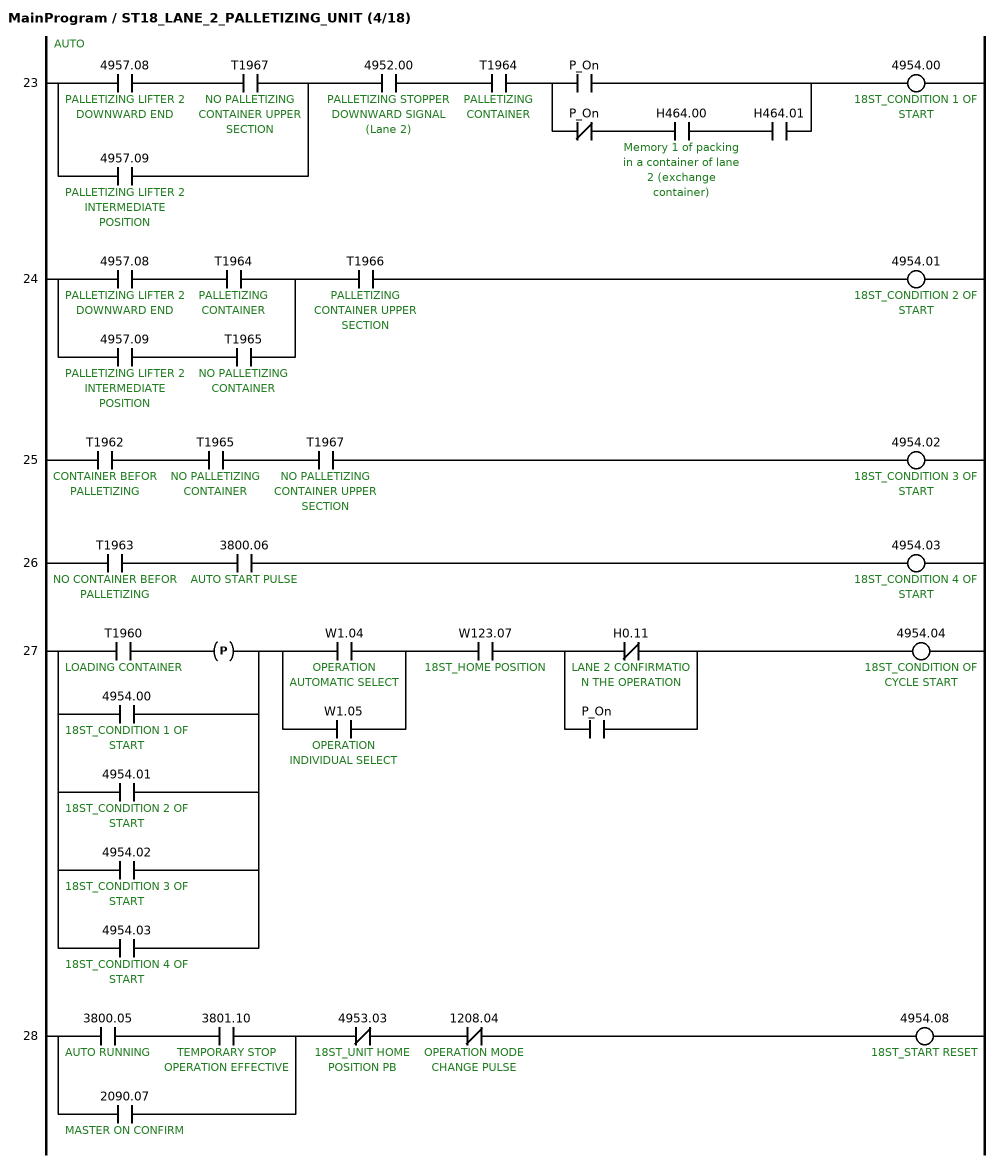
; [picture p672: MainProgram / ST18_LANE_2_PALLETIZING_UNIT, rungs 23-28]
; rung 23: AUTO
LD 4957.08  ; PALLETIZING LIFTER 2 DOWNWARD END
AND T1967  ; NO PALLETIZING CONTAINER UPPER SECTION
OR 4957.09  ; PALLETIZING LIFTER 2 INTERMEDIATE POSITION
AND 4952.00  ; PALLETIZING STOPPER DOWNWARD SIGNAL (Lane 2)
AND T1964  ; PALLETIZING CONTAINER
LD P_On
LDNOT P_On
AND H464.00  ; Memory 1 of packing in a container of lane 2 (exchange container)
AND H464.01
ORLD
ANDLD
OUT 4954.00  ; 18ST_CONDITION 1 OF START
; rung 24
LD 4957.08  ; PALLETIZING LIFTER 2 DOWNWARD END
AND T1964  ; PALLETIZING CONTAINER
LD 4957.09  ; PALLETIZING LIFTER 2 INTERMEDIATE POSITION
AND T1965  ; NO PALLETIZING CONTAINER
ORLD
AND T1966  ; PALLETIZING CONTAINER UPPER SECTION
OUT 4954.01  ; 18ST_CONDITION 2 OF START
; rung 25
LD T1962  ; CONTAINER BEFOR PALLETIZING
AND T1965  ; NO PALLETIZING CONTAINER
AND T1967  ; NO PALLETIZING CONTAINER UPPER SECTION
OUT 4954.02  ; 18ST_CONDITION 3 OF START
; rung 26
LD T1963  ; NO CONTAINER BEFOR PALLETIZING
AND 3800.06  ; AUTO START PULSE
OUT 4954.03  ; 18ST_CONDITION 4 OF START
; rung 27
LD T1960  ; LOADING CONTAINER
UP(521)
OR 4954.00  ; 18ST_CONDITION 1 OF START
OR 4954.01  ; 18ST_CONDITION 2 OF START
OR 4954.02  ; 18ST_CONDITION 3 OF START
OR 4954.03  ; 18ST_CONDITION 4 OF START
LD W1.04  ; OPERATION AUTOMATIC SELECT
OR W1.05  ; OPERATION INDIVIDUAL SELECT
ANDLD
AND W123.07  ; 18ST_HOME POSITION
LDNOT H0.11  ; LANE 2 CONFIRMATION THE OPERATION
OR P_On
ANDLD
OUT 4954.04  ; 18ST_CONDITION OF CYCLE START
; rung 28
LD 3800.05  ; AUTO RUNNING
AND 3801.10  ; TEMPORARY STOP OPERATION EFFECTIVE
OR 2090.07  ; MASTER ON CONFIRM
ANDNOT 4953.03  ; 18ST_UNIT HOME POSITION PB
ANDNOT 1208.04  ; OPERATION MODE CHANGE PULSE
OUT 4954.08  ; 18ST_START RESET

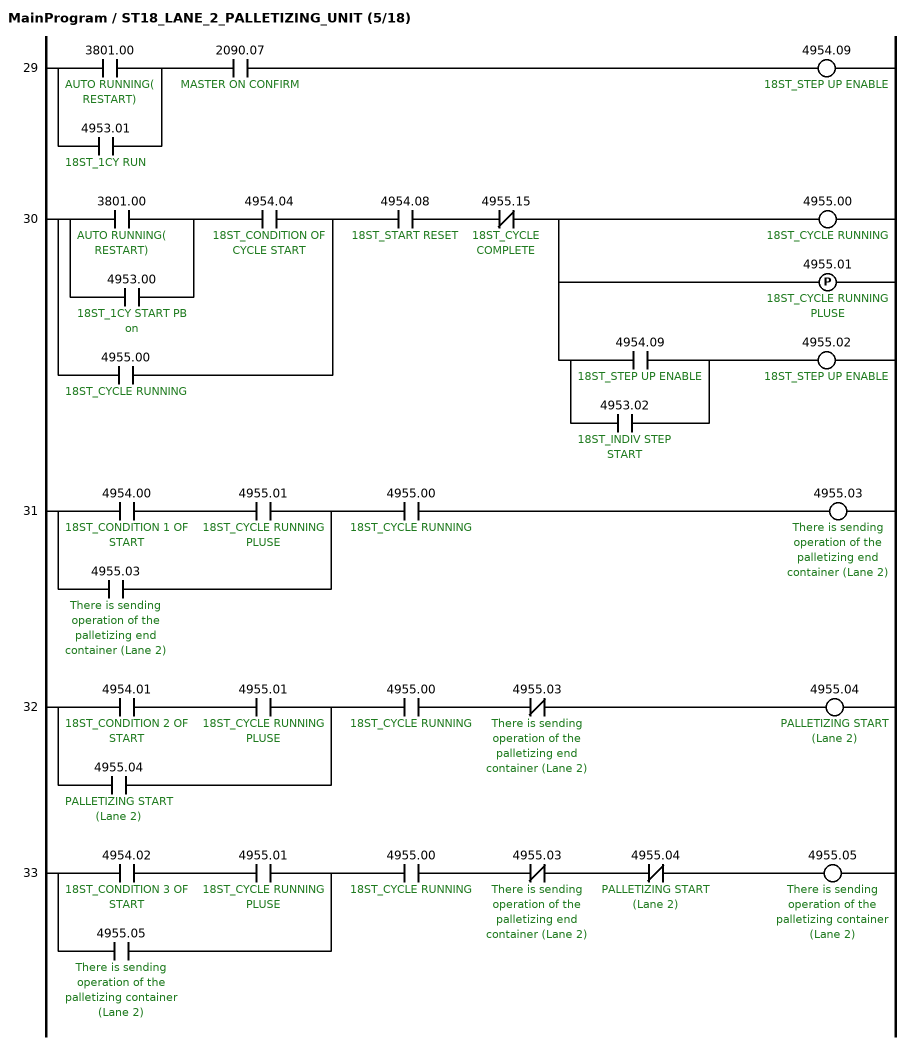
; rung 29
LD 3801.00  ; AUTO RUNNING(RESTART)
OR 4953.01  ; 18ST_1CY RUN
AND 2090.07  ; MASTER ON CONFIRM
OUT 4954.09  ; 18ST_STEP UP ENABLE
; rung 30
LD 3801.00  ; AUTO RUNNING(RESTART)
OR 4953.00  ; 18ST_1CY START PB on
AND 4954.04  ; 18ST_CONDITION OF CYCLE START
OR 4955.00  ; 18ST_CYCLE RUNNING
AND 4954.08  ; 18ST_START RESET
ANDNOT 4955.15  ; 18ST_CYCLE COMPLETE
OUT 4955.00  ; 18ST_CYCLE RUNNING
DIFU(013) 4955.01  ; 18ST_CYCLE RUNNING PLUSE
LD 4954.09  ; 18ST_STEP UP ENABLE
OR 4953.02  ; 18ST_INDIV STEP START
ANDLD
OUT 4955.02  ; 18ST_STEP UP ENABLE
; rung 31
LD 4954.00  ; 18ST_CONDITION 1 OF START
AND 4955.01  ; 18ST_CYCLE RUNNING PLUSE
OR 4955.03  ; There is sending operation of the palletizing end container (Lane 2)
AND 4955.00  ; 18ST_CYCLE RUNNING
OUT 4955.03  ; There is sending operation of the palletizing end container (Lane 2)
; rung 32
LD 4954.01  ; 18ST_CONDITION 2 OF START
AND 4955.01  ; 18ST_CYCLE RUNNING PLUSE
OR 4955.04  ; PALLETIZING START (Lane 2)
AND 4955.00  ; 18ST_CYCLE RUNNING
ANDNOT 4955.03  ; There is sending operation of the palletizing end container (Lane 2)
OUT 4955.04  ; PALLETIZING START (Lane 2)
; rung 33
LD 4954.02  ; 18ST_CONDITION 3 OF START
AND 4955.01  ; 18ST_CYCLE RUNNING PLUSE
OR 4955.05  ; There is sending operation of the palletizing container (Lane 2)
AND 4955.00  ; 18ST_CYCLE RUNNING
ANDNOT 4955.03  ; There is sending operation of the palletizing end container (Lane 2)
ANDNOT 4955.04  ; PALLETIZING START (Lane 2)
OUT 4955.05  ; There is sending operation of the palletizing container (Lane 2)

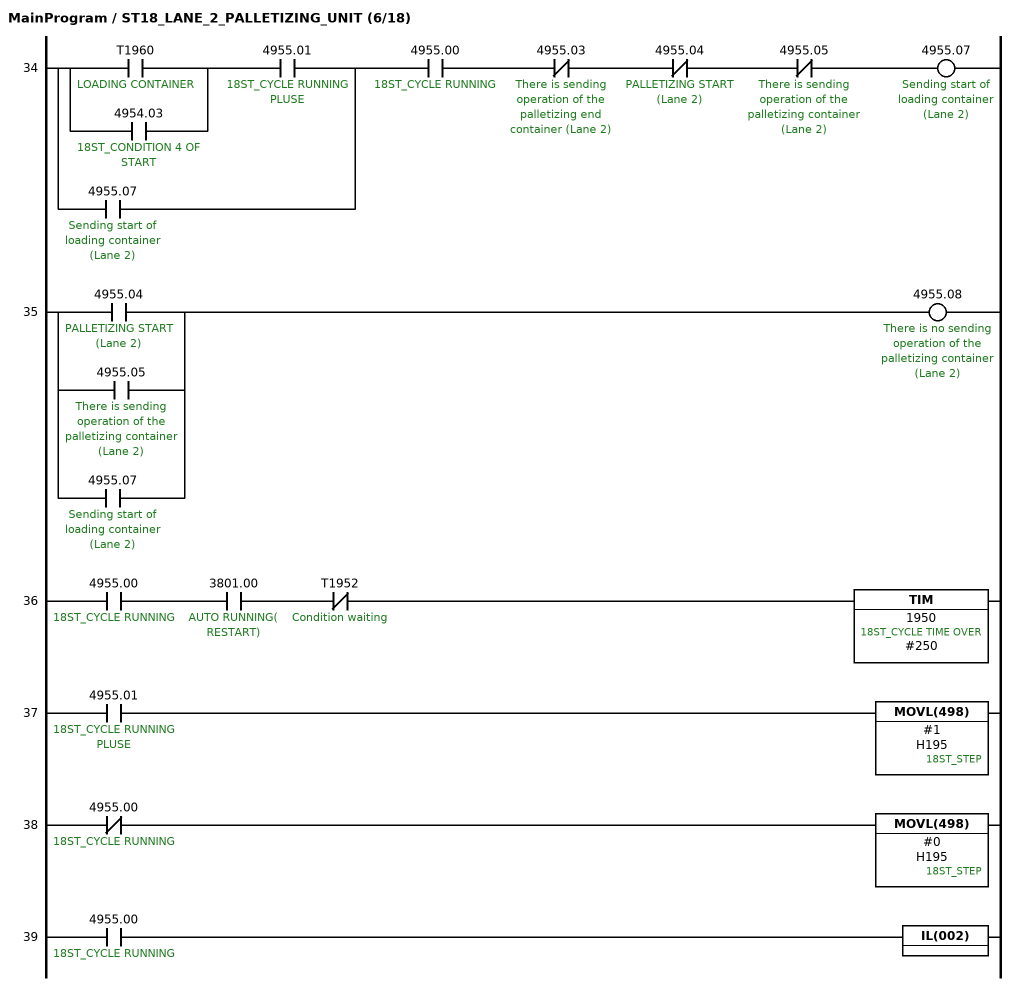
; rung 34
LD T1960  ; LOADING CONTAINER
OR 4954.03  ; 18ST_CONDITION 4 OF START
AND 4955.01  ; 18ST_CYCLE RUNNING PLUSE
OR 4955.07  ; Sending start of loading container (Lane 2)
AND 4955.00  ; 18ST_CYCLE RUNNING
ANDNOT 4955.03  ; There is sending operation of the palletizing end container (Lane 2)
ANDNOT 4955.04  ; PALLETIZING START (Lane 2)
ANDNOT 4955.05  ; There is sending operation of the palletizing container (Lane 2)
OUT 4955.07  ; Sending start of loading container (Lane 2)
; rung 35
LD 4955.04  ; PALLETIZING START (Lane 2)
OR 4955.05  ; There is sending operation of the palletizing container (Lane 2)
OR 4955.07  ; Sending start of loading container (Lane 2)
OUT 4955.08  ; There is no sending operation of the palletizing container (Lane 2)
; rung 36
LD 4955.00  ; 18ST_CYCLE RUNNING
AND 3801.00  ; AUTO RUNNING(RESTART)
ANDNOT T1952  ; Condition waiting
TIM 1950 #250  ; 18ST_CYCLE TIME OVER
; rung 37
LD 4955.01  ; 18ST_CYCLE RUNNING PLUSE
MOVL(498) #1 H195  ; 18ST_STEP
; rung 38
LDNOT 4955.00  ; 18ST_CYCLE RUNNING
MOVL(498) #0 H195  ; 18ST_STEP
; rung 39
LD 4955.00  ; 18ST_CYCLE RUNNING
IL(002)

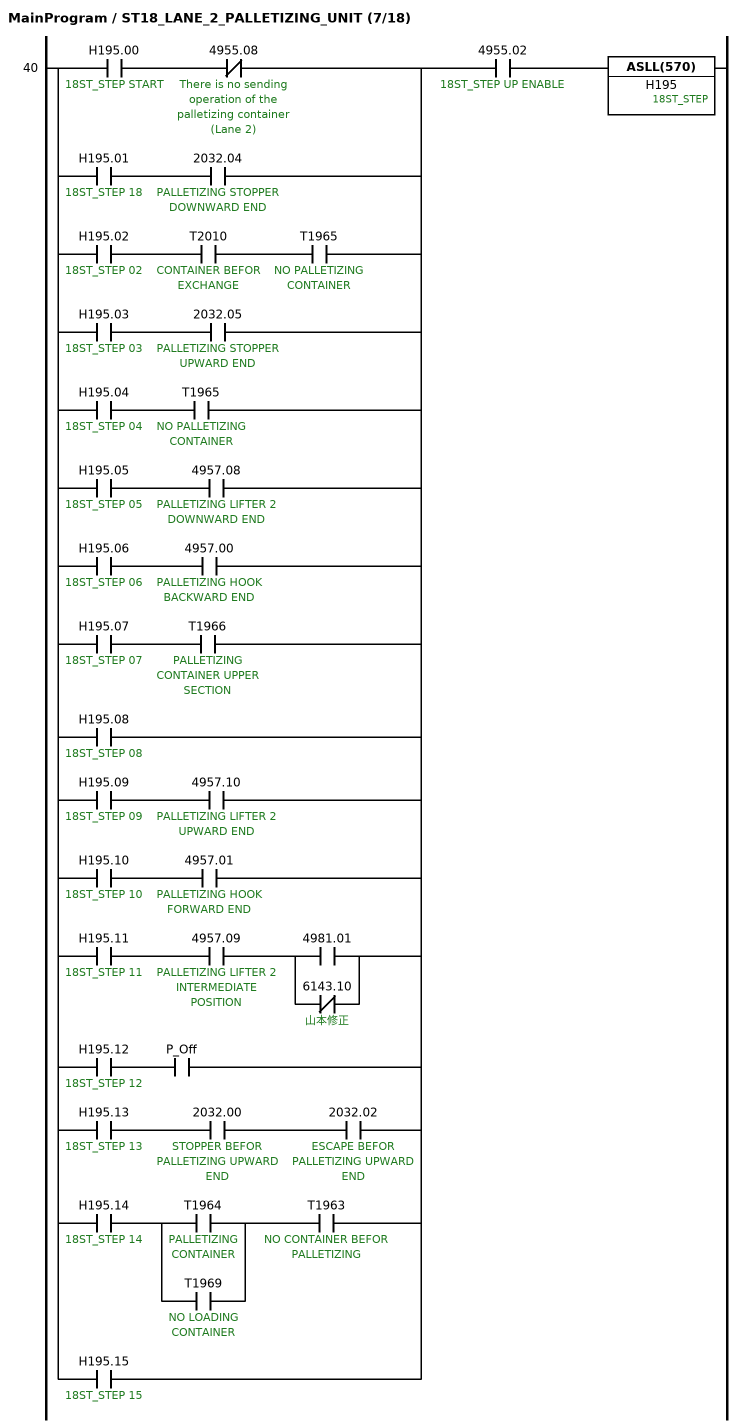
; rung 40
LD H195.00  ; 18ST_STEP START
ANDNOT 4955.08  ; There is no sending operation of the palletizing container (Lane 2)
LD H195.01  ; 18ST_STEP 18
AND 2032.04  ; PALLETIZING STOPPER DOWNWARD END
ORLD
LD H195.02  ; 18ST_STEP 02
AND T2010  ; CONTAINER BEFOR EXCHANGE
AND T1965  ; NO PALLETIZING CONTAINER
ORLD
LD H195.03  ; 18ST_STEP 03
AND 2032.05  ; PALLETIZING STOPPER UPWARD END
ORLD
LD H195.04  ; 18ST_STEP 04
AND T1965  ; NO PALLETIZING CONTAINER
ORLD
LD H195.05  ; 18ST_STEP 05
AND 4957.08  ; PALLETIZING LIFTER 2 DOWNWARD END
ORLD
LD H195.06  ; 18ST_STEP 06
AND 4957.00  ; PALLETIZING HOOK BACKWARD END
ORLD
LD H195.07  ; 18ST_STEP 07
AND T1966  ; PALLETIZING CONTAINER UPPER SECTION
ORLD
OR H195.08  ; 18ST_STEP 08
LD H195.09  ; 18ST_STEP 09
AND 4957.10  ; PALLETIZING LIFTER 2 UPWARD END
ORLD
LD H195.10  ; 18ST_STEP 10
AND 4957.01  ; PALLETIZING HOOK FORWARD END
ORLD
LD H195.11  ; 18ST_STEP 11
AND 4957.09  ; PALLETIZING LIFTER 2 INTERMEDIATE POSITION
LD 4981.01
ORNOT 6143.10  ; 山本修正
ANDLD
ORLD
LD H195.12  ; 18ST_STEP 12
AND P_Off
ORLD
LD H195.13  ; 18ST_STEP 13
AND 2032.00  ; STOPPER BEFOR PALLETIZING UPWARD END
AND 2032.02  ; ESCAPE BEFOR PALLETIZING UPWARD END
ORLD
LD H195.14  ; 18ST_STEP 14
LD T1964  ; PALLETIZING CONTAINER
OR T1969  ; NO LOADING CONTAINER
ANDLD
AND T1963  ; NO CONTAINER BEFOR PALLETIZING
ORLD
OR H195.15  ; 18ST_STEP 15
AND 4955.02  ; 18ST_STEP UP ENABLE
ASLL(570) H195  ; 18ST_STEP

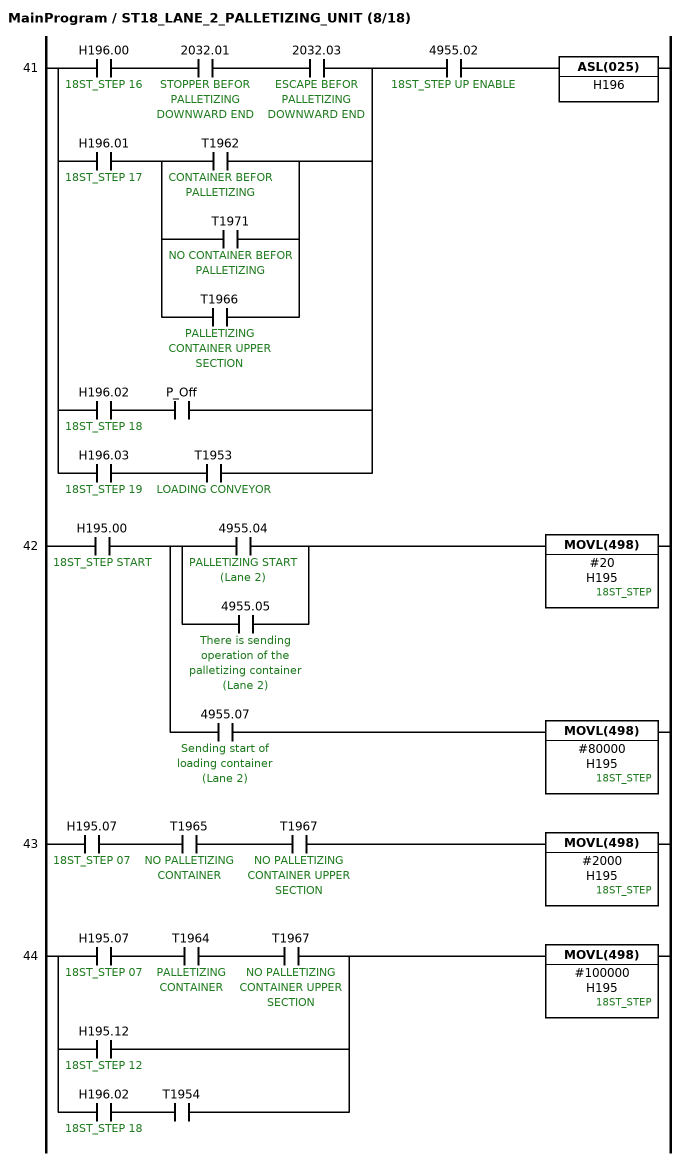
; rung 41
LD H196.00  ; 18ST_STEP 16
AND 2032.01  ; STOPPER BEFOR PALLETIZING DOWNWARD END
AND 2032.03  ; ESCAPE BEFOR PALLETIZING DOWNWARD END
LD H196.01  ; 18ST_STEP 17
LD T1962  ; CONTAINER BEFOR PALLETIZING
OR T1971  ; NO CONTAINER BEFOR PALLETIZING
OR T1966  ; PALLETIZING CONTAINER UPPER SECTION
ANDLD
ORLD
LD H196.02  ; 18ST_STEP 18
AND P_Off
ORLD
LD H196.03  ; 18ST_STEP 19
AND T1953  ; LOADING CONVEYOR
ORLD
AND 4955.02  ; 18ST_STEP UP ENABLE
ASL(025) H196
; rung 42
LD H195.00  ; 18ST_STEP START
OUT TR0
LD 4955.04  ; PALLETIZING START (Lane 2)
OR 4955.05  ; There is sending operation of the palletizing container (Lane 2)
ANDLD
MOVL(498) #20 H195  ; 18ST_STEP
LD TR0
AND 4955.07  ; Sending start of loading container (Lane 2)
MOVL(498) #80000 H195  ; 18ST_STEP
; rung 43
LD H195.07  ; 18ST_STEP 07
AND T1965  ; NO PALLETIZING CONTAINER
AND T1967  ; NO PALLETIZING CONTAINER UPPER SECTION
MOVL(498) #2000 H195  ; 18ST_STEP
; rung 44
LD H195.07  ; 18ST_STEP 07
AND T1964  ; PALLETIZING CONTAINER
AND T1967  ; NO PALLETIZING CONTAINER UPPER SECTION
OR H195.12  ; 18ST_STEP 12
LD H196.02  ; 18ST_STEP 18
AND T1954
ORLD
MOVL(498) #100000 H195  ; 18ST_STEP

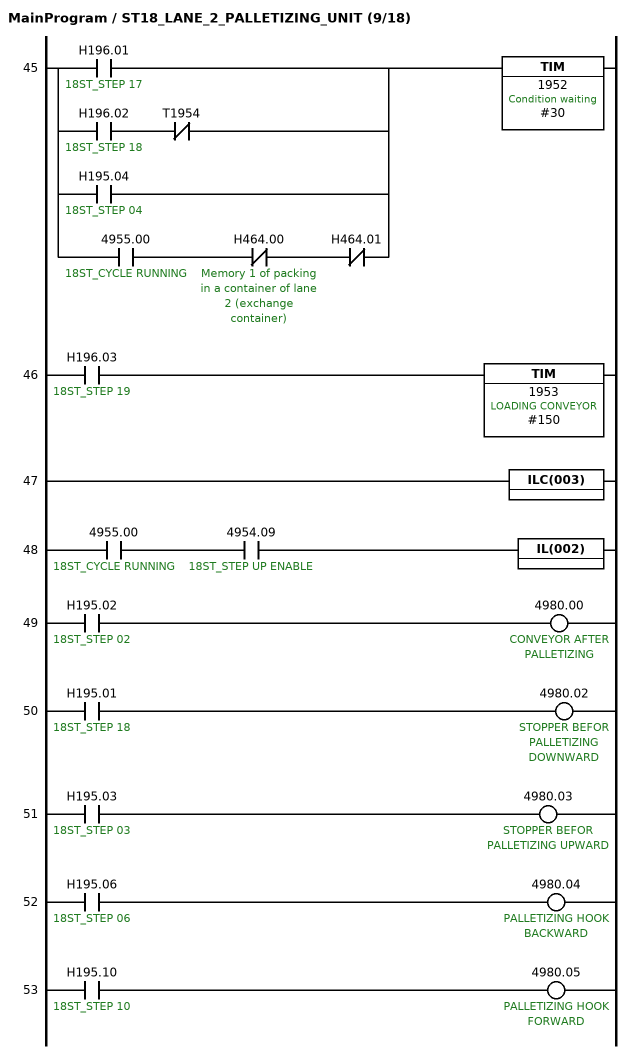
; rung 45
LD H196.01  ; 18ST_STEP 17
LD H196.02  ; 18ST_STEP 18
ANDNOT T1954
ORLD
OR H195.04  ; 18ST_STEP 04
LD 4955.00  ; 18ST_CYCLE RUNNING
ANDNOT H464.00  ; Memory 1 of packing in a container of lane 2 (exchange container)
ANDNOT H464.01
ORLD
TIM 1952 #30  ; Condition waiting
; rung 46
LD H196.03  ; 18ST_STEP 19
TIM 1953 #150  ; LOADING CONVEYOR
; rung 47
ILC(003)
; rung 48
LD 4955.00  ; 18ST_CYCLE RUNNING
AND 4954.09  ; 18ST_STEP UP ENABLE
IL(002)
; rung 49
LD H195.02  ; 18ST_STEP 02
OUT 4980.00  ; CONVEYOR AFTER PALLETIZING
; rung 50
LD H195.01  ; 18ST_STEP 18
OUT 4980.02  ; STOPPER BEFOR PALLETIZING DOWNWARD
; rung 51
LD H195.03  ; 18ST_STEP 03
OUT 4980.03  ; STOPPER BEFOR PALLETIZING UPWARD
; rung 52
LD H195.06  ; 18ST_STEP 06
OUT 4980.04  ; PALLETIZING HOOK BACKWARD
; rung 53
LD H195.10  ; 18ST_STEP 10
OUT 4980.05  ; PALLETIZING HOOK FORWARD

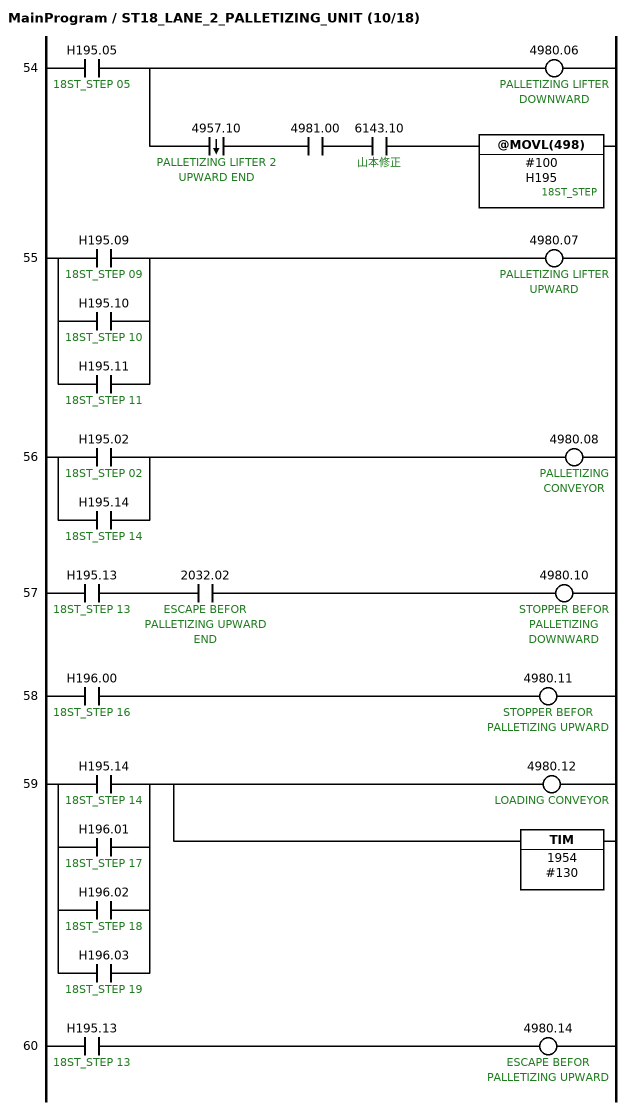
; rung 54
LD H195.05  ; 18ST_STEP 05
OUT 4980.06  ; PALLETIZING LIFTER DOWNWARD
%AND 4957.10  ; PALLETIZING LIFTER 2 UPWARD END
AND 4981.00
AND 6143.10  ; 山本修正
@MOVL(498) #100 H195  ; 18ST_STEP
; rung 55
LD H195.09  ; 18ST_STEP 09
OR H195.10  ; 18ST_STEP 10
OR H195.11  ; 18ST_STEP 11
OUT 4980.07  ; PALLETIZING LIFTER UPWARD
; rung 56
LD H195.02  ; 18ST_STEP 02
OR H195.14  ; 18ST_STEP 14
OUT 4980.08  ; PALLETIZING CONVEYOR
; rung 57
LD H195.13  ; 18ST_STEP 13
AND 2032.02  ; ESCAPE BEFOR PALLETIZING UPWARD END
OUT 4980.10  ; STOPPER BEFOR PALLETIZING DOWNWARD
; rung 58
LD H196.00  ; 18ST_STEP 16
OUT 4980.11  ; STOPPER BEFOR PALLETIZING UPWARD
; rung 59
LD H195.14  ; 18ST_STEP 14
OR H196.01  ; 18ST_STEP 17
OR H196.02  ; 18ST_STEP 18
OR H196.03  ; 18ST_STEP 19
OUT 4980.12  ; LOADING CONVEYOR
TIM 1954 #130
; rung 60
LD H195.13  ; 18ST_STEP 13
OUT 4980.14  ; ESCAPE BEFOR PALLETIZING UPWARD

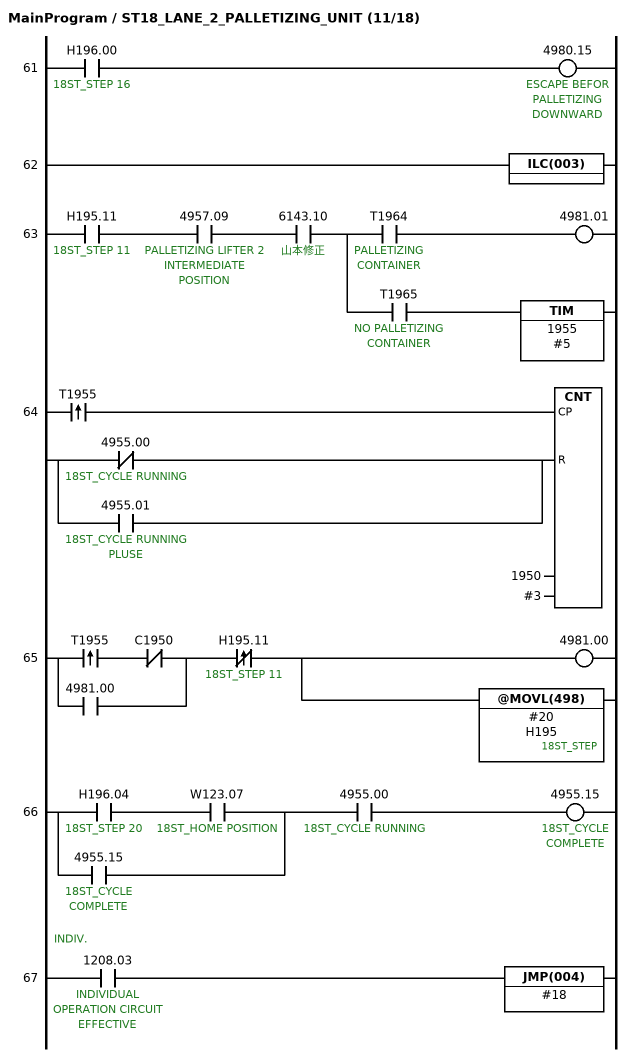
; rung 61
LD H196.00  ; 18ST_STEP 16
OUT 4980.15  ; ESCAPE BEFOR PALLETIZING DOWNWARD
; rung 62
ILC(003)
; rung 63
LD H195.11  ; 18ST_STEP 11
AND 4957.09  ; PALLETIZING LIFTER 2 INTERMEDIATE POSITION
AND 6143.10  ; 山本修正
OUT TR0
AND T1964  ; PALLETIZING CONTAINER
OUT 4981.01
LD TR0
AND T1965  ; NO PALLETIZING CONTAINER
TIM 1955 #5
; rung 64
@LD T1955
LDNOT 4955.00  ; 18ST_CYCLE RUNNING
OR 4955.01  ; 18ST_CYCLE RUNNING PLUSE
CNT 1950 #3
; rung 65
@LD T1955
ANDNOT C1950
OR 4981.00
@ANDNOT H195.11  ; 18ST_STEP 11
OUT 4981.00
@MOVL(498) #20 H195  ; 18ST_STEP
; rung 66
LD H196.04  ; 18ST_STEP 20
AND W123.07  ; 18ST_HOME POSITION
OR 4955.15  ; 18ST_CYCLE COMPLETE
AND 4955.00  ; 18ST_CYCLE RUNNING
OUT 4955.15  ; 18ST_CYCLE COMPLETE
; rung 67: INDIV.
LD 1208.03  ; INDIVIDUAL OPERATION CIRCUIT EFFECTIVE
JMP(004) #18

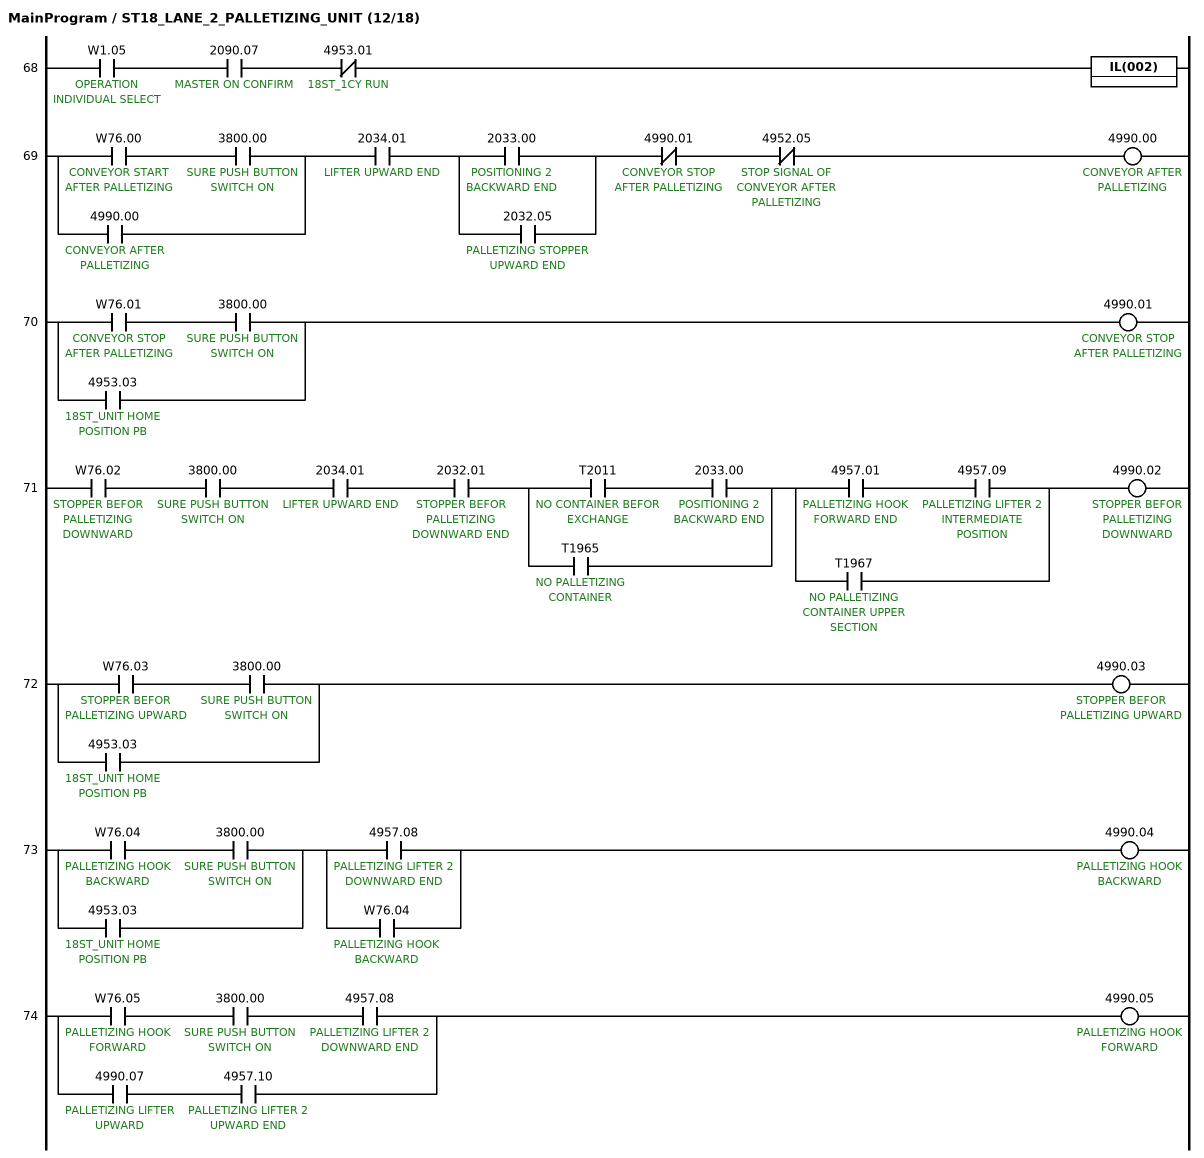
; rung 68
LD W1.05  ; OPERATION INDIVIDUAL SELECT
AND 2090.07  ; MASTER ON CONFIRM
ANDNOT 4953.01  ; 18ST_1CY RUN
IL(002)
; rung 69
LD W76.00  ; CONVEYOR START AFTER PALLETIZING
AND 3800.00  ; SURE PUSH BUTTON SWITCH ON
OR 4990.00  ; CONVEYOR AFTER PALLETIZING
AND 2034.01  ; LIFTER UPWARD END
LD 2033.00  ; POSITIONING 2 BACKWARD END
OR 2032.05  ; PALLETIZING STOPPER UPWARD END
ANDLD
ANDNOT 4990.01  ; CONVEYOR STOP AFTER PALLETIZING
ANDNOT 4952.05  ; STOP SIGNAL OF CONVEYOR AFTER PALLETIZING
OUT 4990.00  ; CONVEYOR AFTER PALLETIZING
; rung 70
LD W76.01  ; CONVEYOR STOP AFTER PALLETIZING
AND 3800.00  ; SURE PUSH BUTTON SWITCH ON
OR 4953.03  ; 18ST_UNIT HOME POSITION PB
OUT 4990.01  ; CONVEYOR STOP AFTER PALLETIZING
; rung 71
LD W76.02  ; STOPPER BEFOR PALLETIZING DOWNWARD
AND 3800.00  ; SURE PUSH BUTTON SWITCH ON
AND 2034.01  ; LIFTER UPWARD END
AND 2032.01  ; STOPPER BEFOR PALLETIZING DOWNWARD END
LD T2011  ; NO CONTAINER BEFOR EXCHANGE
AND 2033.00  ; POSITIONING 2 BACKWARD END
OR T1965  ; NO PALLETIZING CONTAINER
ANDLD
LD 4957.01  ; PALLETIZING HOOK FORWARD END
AND 4957.09  ; PALLETIZING LIFTER 2 INTERMEDIATE POSITION
OR T1967  ; NO PALLETIZING CONTAINER UPPER SECTION
ANDLD
OUT 4990.02  ; STOPPER BEFOR PALLETIZING DOWNWARD
; rung 72
LD W76.03  ; STOPPER BEFOR PALLETIZING UPWARD
AND 3800.00  ; SURE PUSH BUTTON SWITCH ON
OR 4953.03  ; 18ST_UNIT HOME POSITION PB
OUT 4990.03  ; STOPPER BEFOR PALLETIZING UPWARD
; rung 73
LD W76.04  ; PALLETIZING HOOK BACKWARD
AND 3800.00  ; SURE PUSH BUTTON SWITCH ON
OR 4953.03  ; 18ST_UNIT HOME POSITION PB
LD 4957.08  ; PALLETIZING LIFTER 2 DOWNWARD END
OR W76.04  ; PALLETIZING HOOK BACKWARD
ANDLD
OUT 4990.04  ; PALLETIZING HOOK BACKWARD
; rung 74
LD W76.05  ; PALLETIZING HOOK FORWARD
AND 3800.00  ; SURE PUSH BUTTON SWITCH ON
AND 4957.08  ; PALLETIZING LIFTER 2 DOWNWARD END
LD 4990.07  ; PALLETIZING LIFTER UPWARD
AND 4957.10  ; PALLETIZING LIFTER 2 UPWARD END
ORLD
OUT 4990.05  ; PALLETIZING HOOK FORWARD

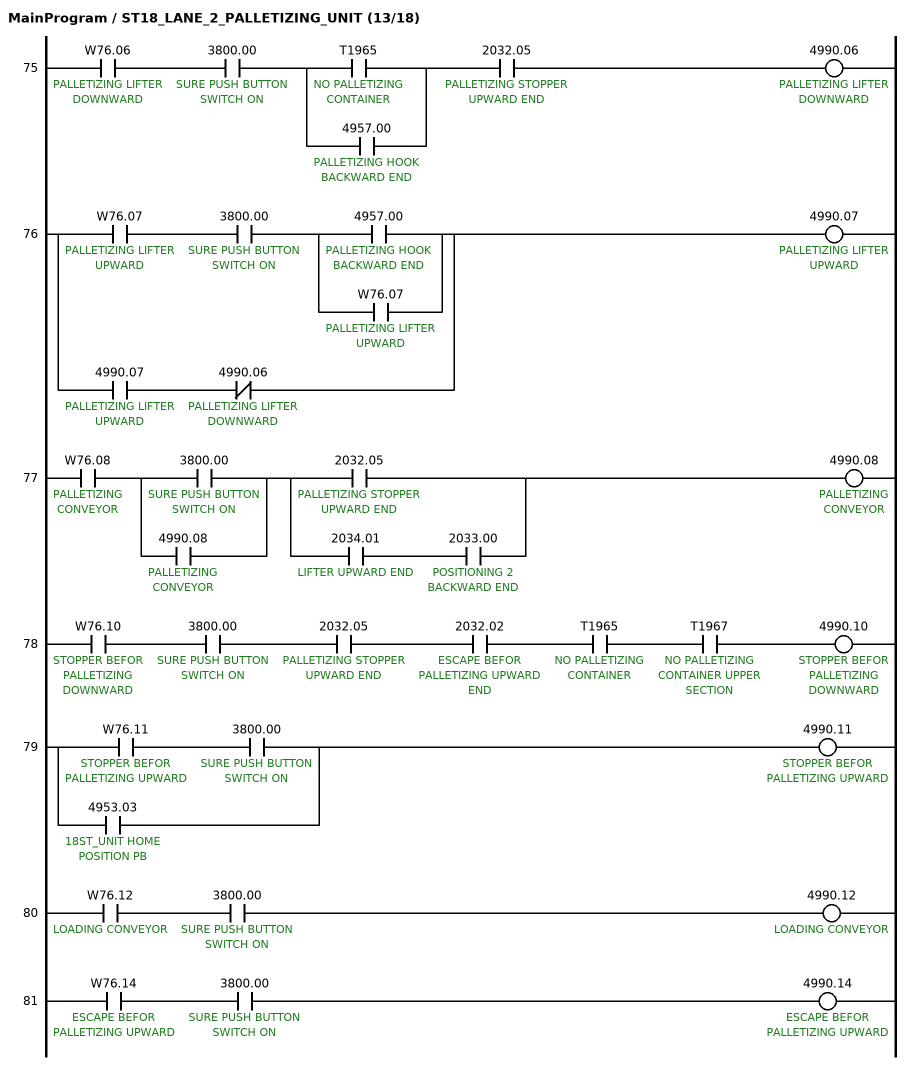
; rung 75
LD W76.06  ; PALLETIZING LIFTER DOWNWARD
AND 3800.00  ; SURE PUSH BUTTON SWITCH ON
LD T1965  ; NO PALLETIZING CONTAINER
OR 4957.00  ; PALLETIZING HOOK BACKWARD END
ANDLD
AND 2032.05  ; PALLETIZING STOPPER UPWARD END
OUT 4990.06  ; PALLETIZING LIFTER DOWNWARD
; rung 76
LD W76.07  ; PALLETIZING LIFTER UPWARD
AND 3800.00  ; SURE PUSH BUTTON SWITCH ON
LD 4957.00  ; PALLETIZING HOOK BACKWARD END
OR W76.07  ; PALLETIZING LIFTER UPWARD
ANDLD
LD 4990.07  ; PALLETIZING LIFTER UPWARD
ANDNOT 4990.06  ; PALLETIZING LIFTER DOWNWARD
ORLD
OUT 4990.07  ; PALLETIZING LIFTER UPWARD
; rung 77
LD W76.08  ; PALLETIZING CONVEYOR
LD 3800.00  ; SURE PUSH BUTTON SWITCH ON
OR 4990.08  ; PALLETIZING CONVEYOR
ANDLD
LD 2032.05  ; PALLETIZING STOPPER UPWARD END
LD 2034.01  ; LIFTER UPWARD END
AND 2033.00  ; POSITIONING 2 BACKWARD END
ORLD
ANDLD
OUT 4990.08  ; PALLETIZING CONVEYOR
; rung 78
LD W76.10  ; STOPPER BEFOR PALLETIZING DOWNWARD
AND 3800.00  ; SURE PUSH BUTTON SWITCH ON
AND 2032.05  ; PALLETIZING STOPPER UPWARD END
AND 2032.02  ; ESCAPE BEFOR PALLETIZING UPWARD END
AND T1965  ; NO PALLETIZING CONTAINER
AND T1967  ; NO PALLETIZING CONTAINER UPPER SECTION
OUT 4990.10  ; STOPPER BEFOR PALLETIZING DOWNWARD
; rung 79
LD W76.11  ; STOPPER BEFOR PALLETIZING UPWARD
AND 3800.00  ; SURE PUSH BUTTON SWITCH ON
OR 4953.03  ; 18ST_UNIT HOME POSITION PB
OUT 4990.11  ; STOPPER BEFOR PALLETIZING UPWARD
; rung 80
LD W76.12  ; LOADING CONVEYOR
AND 3800.00  ; SURE PUSH BUTTON SWITCH ON
OUT 4990.12  ; LOADING CONVEYOR
; rung 81
LD W76.14  ; ESCAPE BEFOR PALLETIZING UPWARD
AND 3800.00  ; SURE PUSH BUTTON SWITCH ON
OUT 4990.14  ; ESCAPE BEFOR PALLETIZING UPWARD

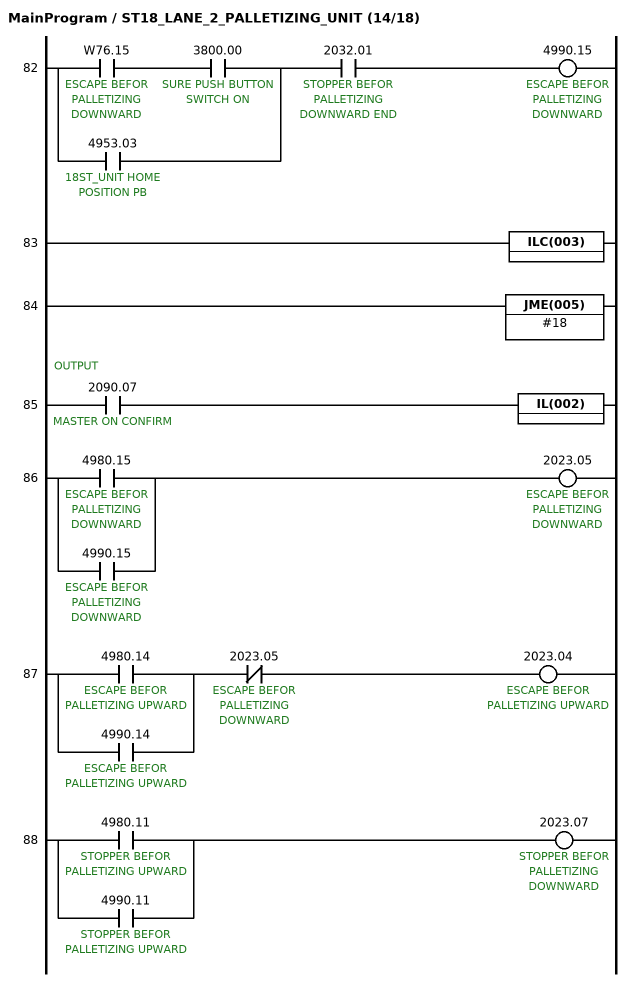
; rung 82
LD W76.15  ; ESCAPE BEFOR PALLETIZING DOWNWARD
AND 3800.00  ; SURE PUSH BUTTON SWITCH ON
OR 4953.03  ; 18ST_UNIT HOME POSITION PB
AND 2032.01  ; STOPPER BEFOR PALLETIZING DOWNWARD END
OUT 4990.15  ; ESCAPE BEFOR PALLETIZING DOWNWARD
; rung 83
ILC(003)
; rung 84
JME(005) #18
; rung 85: OUTPUT
LD 2090.07  ; MASTER ON CONFIRM
IL(002)
; rung 86
LD 4980.15  ; ESCAPE BEFOR PALLETIZING DOWNWARD
OR 4990.15  ; ESCAPE BEFOR PALLETIZING DOWNWARD
OUT 2023.05  ; ESCAPE BEFOR PALLETIZING DOWNWARD
; rung 87
LD 4980.14  ; ESCAPE BEFOR PALLETIZING UPWARD
OR 4990.14  ; ESCAPE BEFOR PALLETIZING UPWARD
ANDNOT 2023.05  ; ESCAPE BEFOR PALLETIZING DOWNWARD
OUT 2023.04  ; ESCAPE BEFOR PALLETIZING UPWARD
; rung 88
LD 4980.11  ; STOPPER BEFOR PALLETIZING UPWARD
OR 4990.11  ; STOPPER BEFOR PALLETIZING UPWARD
OUT 2023.07  ; STOPPER BEFOR PALLETIZING DOWNWARD

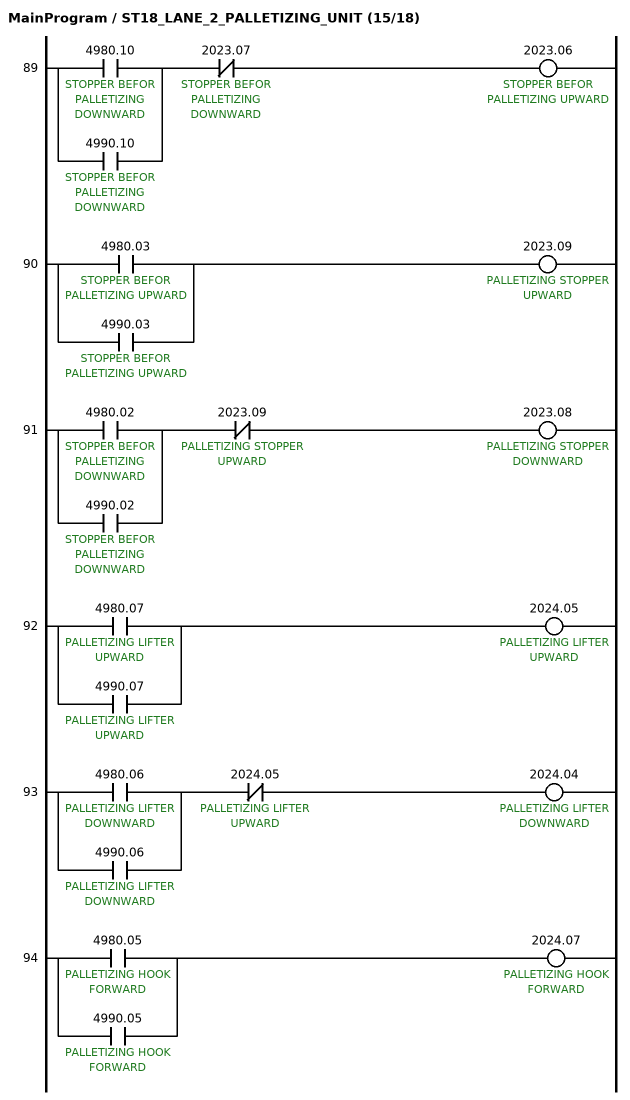
; rung 89
LD 4980.10  ; STOPPER BEFOR PALLETIZING DOWNWARD
OR 4990.10  ; STOPPER BEFOR PALLETIZING DOWNWARD
ANDNOT 2023.07  ; STOPPER BEFOR PALLETIZING DOWNWARD
OUT 2023.06  ; STOPPER BEFOR PALLETIZING UPWARD
; rung 90
LD 4980.03  ; STOPPER BEFOR PALLETIZING UPWARD
OR 4990.03  ; STOPPER BEFOR PALLETIZING UPWARD
OUT 2023.09  ; PALLETIZING STOPPER UPWARD
; rung 91
LD 4980.02  ; STOPPER BEFOR PALLETIZING DOWNWARD
OR 4990.02  ; STOPPER BEFOR PALLETIZING DOWNWARD
ANDNOT 2023.09  ; PALLETIZING STOPPER UPWARD
OUT 2023.08  ; PALLETIZING STOPPER DOWNWARD
; rung 92
LD 4980.07  ; PALLETIZING LIFTER UPWARD
OR 4990.07  ; PALLETIZING LIFTER UPWARD
OUT 2024.05  ; PALLETIZING LIFTER UPWARD
; rung 93
LD 4980.06  ; PALLETIZING LIFTER DOWNWARD
OR 4990.06  ; PALLETIZING LIFTER DOWNWARD
ANDNOT 2024.05  ; PALLETIZING LIFTER UPWARD
OUT 2024.04  ; PALLETIZING LIFTER DOWNWARD
; rung 94
LD 4980.05  ; PALLETIZING HOOK FORWARD
OR 4990.05  ; PALLETIZING HOOK FORWARD
OUT 2024.07  ; PALLETIZING HOOK FORWARD

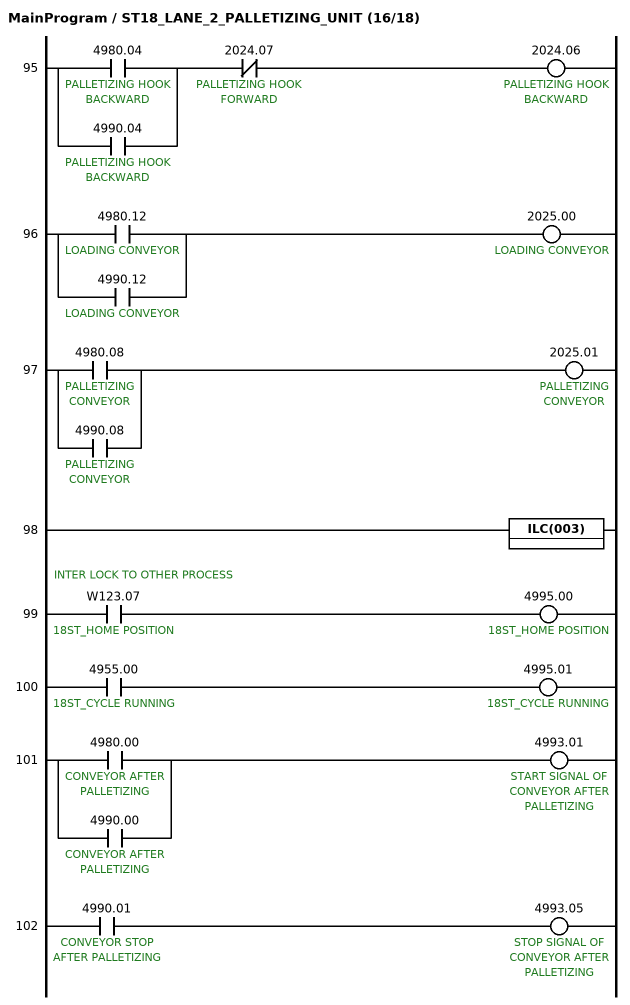
; rung 95
LD 4980.04  ; PALLETIZING HOOK BACKWARD
OR 4990.04  ; PALLETIZING HOOK BACKWARD
ANDNOT 2024.07  ; PALLETIZING HOOK FORWARD
OUT 2024.06  ; PALLETIZING HOOK BACKWARD
; rung 96
LD 4980.12  ; LOADING CONVEYOR
OR 4990.12  ; LOADING CONVEYOR
OUT 2025.00  ; LOADING CONVEYOR
; rung 97
LD 4980.08  ; PALLETIZING CONVEYOR
OR 4990.08  ; PALLETIZING CONVEYOR
OUT 2025.01  ; PALLETIZING CONVEYOR
; rung 98
ILC(003)
; rung 99: INTER LOCK TO OTHER PROCESS
LD W123.07  ; 18ST_HOME POSITION
OUT 4995.00  ; 18ST_HOME POSITION
; rung 100
LD 4955.00  ; 18ST_CYCLE RUNNING
OUT 4995.01  ; 18ST_CYCLE RUNNING
; rung 101
LD 4980.00  ; CONVEYOR AFTER PALLETIZING
OR 4990.00  ; CONVEYOR AFTER PALLETIZING
OUT 4993.01  ; START SIGNAL OF CONVEYOR AFTER PALLETIZING
; rung 102
LD 4990.01  ; CONVEYOR STOP AFTER PALLETIZING
OUT 4993.05  ; STOP SIGNAL OF CONVEYOR AFTER PALLETIZING

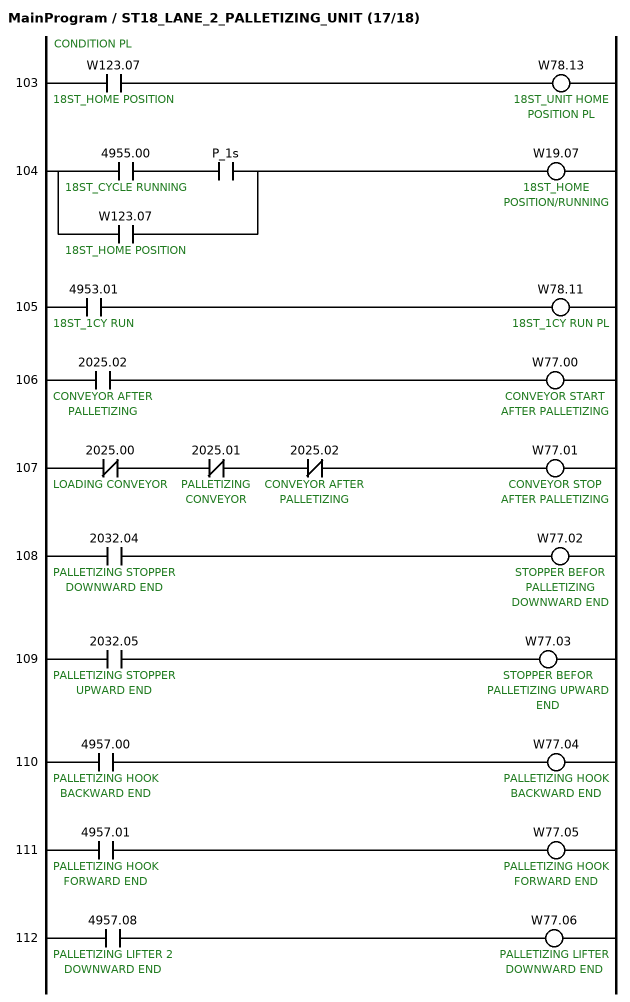
; rung 103: CONDITION PL
LD W123.07  ; 18ST_HOME POSITION
OUT W78.13  ; 18ST_UNIT HOME POSITION PL
; rung 104
LD 4955.00  ; 18ST_CYCLE RUNNING
AND P_1s
OR W123.07  ; 18ST_HOME POSITION
OUT W19.07  ; 18ST_HOME POSITION/RUNNING
; rung 105
LD 4953.01  ; 18ST_1CY RUN
OUT W78.11  ; 18ST_1CY RUN PL
; rung 106
LD 2025.02  ; CONVEYOR AFTER PALLETIZING
OUT W77.00  ; CONVEYOR START AFTER PALLETIZING
; rung 107
LDNOT 2025.00  ; LOADING CONVEYOR
ANDNOT 2025.01  ; PALLETIZING CONVEYOR
ANDNOT 2025.02  ; CONVEYOR AFTER PALLETIZING
OUT W77.01  ; CONVEYOR STOP AFTER PALLETIZING
; rung 108
LD 2032.04  ; PALLETIZING STOPPER DOWNWARD END
OUT W77.02  ; STOPPER BEFOR PALLETIZING DOWNWARD END
; rung 109
LD 2032.05  ; PALLETIZING STOPPER UPWARD END
OUT W77.03  ; STOPPER BEFOR PALLETIZING UPWARD END
; rung 110
LD 4957.00  ; PALLETIZING HOOK BACKWARD END
OUT W77.04  ; PALLETIZING HOOK BACKWARD END
; rung 111
LD 4957.01  ; PALLETIZING HOOK FORWARD END
OUT W77.05  ; PALLETIZING HOOK FORWARD END
; rung 112
LD 4957.08  ; PALLETIZING LIFTER 2 DOWNWARD END
OUT W77.06  ; PALLETIZING LIFTER DOWNWARD END

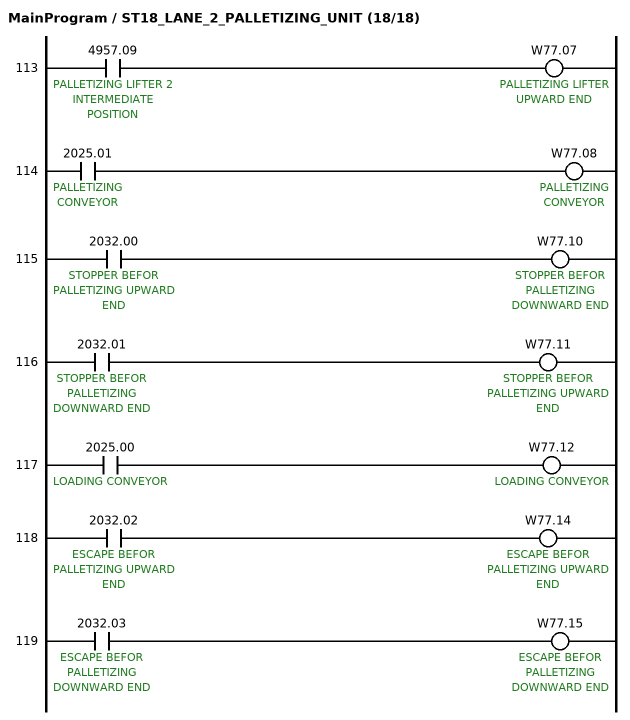
; rung 113
LD 4957.09  ; PALLETIZING LIFTER 2 INTERMEDIATE POSITION
OUT W77.07  ; PALLETIZING LIFTER UPWARD END
; rung 114
LD 2025.01  ; PALLETIZING CONVEYOR
OUT W77.08  ; PALLETIZING CONVEYOR
; rung 115
LD 2032.00  ; STOPPER BEFOR PALLETIZING UPWARD END
OUT W77.10  ; STOPPER BEFOR PALLETIZING DOWNWARD END
; rung 116
LD 2032.01  ; STOPPER BEFOR PALLETIZING DOWNWARD END
OUT W77.11  ; STOPPER BEFOR PALLETIZING UPWARD END
; rung 117
LD 2025.00  ; LOADING CONVEYOR
OUT W77.12  ; LOADING CONVEYOR
; rung 118
LD 2032.02  ; ESCAPE BEFOR PALLETIZING UPWARD END
OUT W77.14  ; ESCAPE BEFOR PALLETIZING UPWARD END
; rung 119
LD 2032.03  ; ESCAPE BEFOR PALLETIZING DOWNWARD END
OUT W77.15  ; ESCAPE BEFOR PALLETIZING DOWNWARD END
; rung 120

### Section ST19_LANE_2_SUPPLYING_UNIT

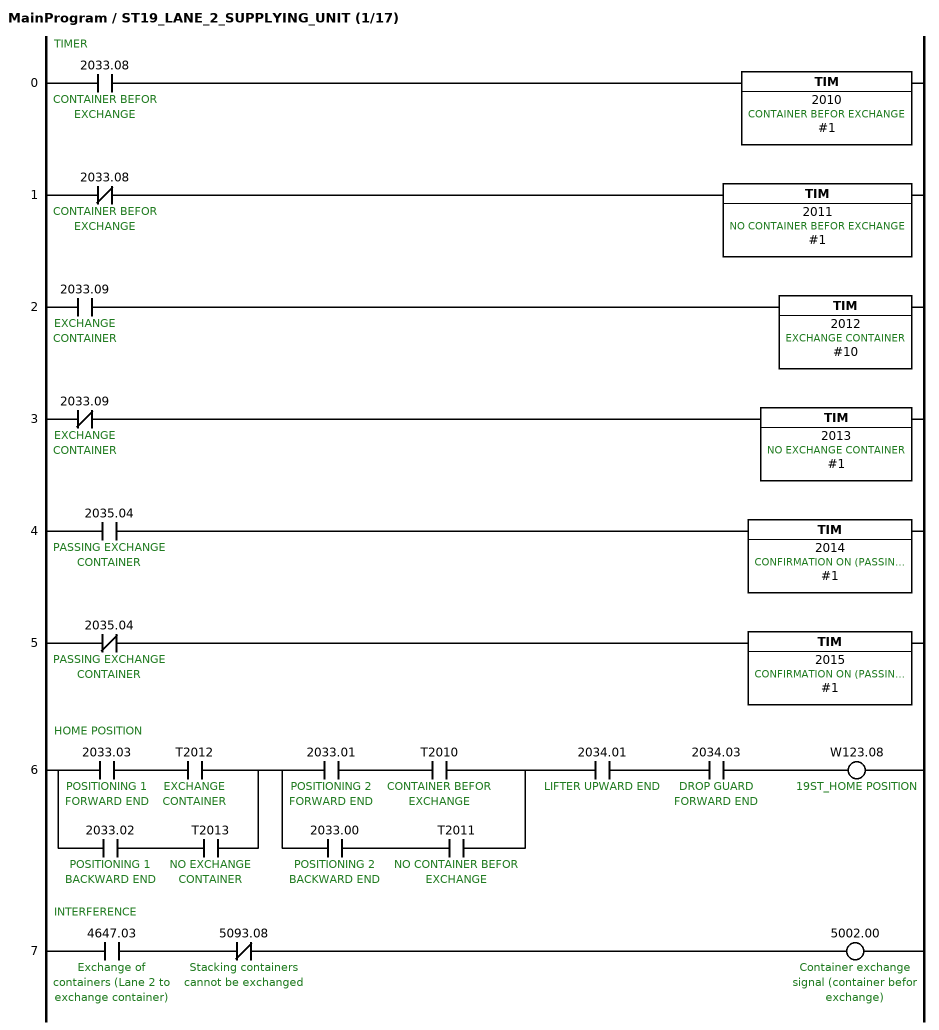
; rung 0: TIMER
LD 2033.08  ; CONTAINER BEFOR EXCHANGE
TIM 2010 #1  ; CONTAINER BEFOR EXCHANGE
; rung 1
LDNOT 2033.08  ; CONTAINER BEFOR EXCHANGE
TIM 2011 #1  ; NO CONTAINER BEFOR EXCHANGE
; rung 2
LD 2033.09  ; EXCHANGE CONTAINER
TIM 2012 #10  ; EXCHANGE CONTAINER
; rung 3
LDNOT 2033.09  ; EXCHANGE CONTAINER
TIM 2013 #1  ; NO EXCHANGE CONTAINER
; rung 4
LD 2035.04  ; PASSING EXCHANGE CONTAINER
TIM 2014 #1  ; CONFIRMATION ON (PASSING EXCHANGE CONTAINER)
; rung 5
LDNOT 2035.04  ; PASSING EXCHANGE CONTAINER
TIM 2015 #1  ; CONFIRMATION ON (PASSING EXCHANGE CONTAINER)
; rung 6: HOME POSITION
LD 2033.03  ; POSITIONING 1 FORWARD END
AND T2012  ; EXCHANGE CONTAINER
LD 2033.02  ; POSITIONING 1 BACKWARD END
AND T2013  ; NO EXCHANGE CONTAINER
ORLD
LD 2033.01  ; POSITIONING 2 FORWARD END
AND T2010  ; CONTAINER BEFOR EXCHANGE
LD 2033.00  ; POSITIONING 2 BACKWARD END
AND T2011  ; NO CONTAINER BEFOR EXCHANGE
ORLD
ANDLD
AND 2034.01  ; LIFTER UPWARD END
AND 2034.03  ; DROP GUARD FORWARD END
OUT W123.08  ; 19ST_HOME POSITION
; rung 7: INTERFERENCE
LD 4647.03  ; Exchange of containers (Lane 2 to exchange container)
ANDNOT 5093.08  ; Stacking containers cannot be exchanged
OUT 5002.00  ; Container exchange signal (container befor exchange)

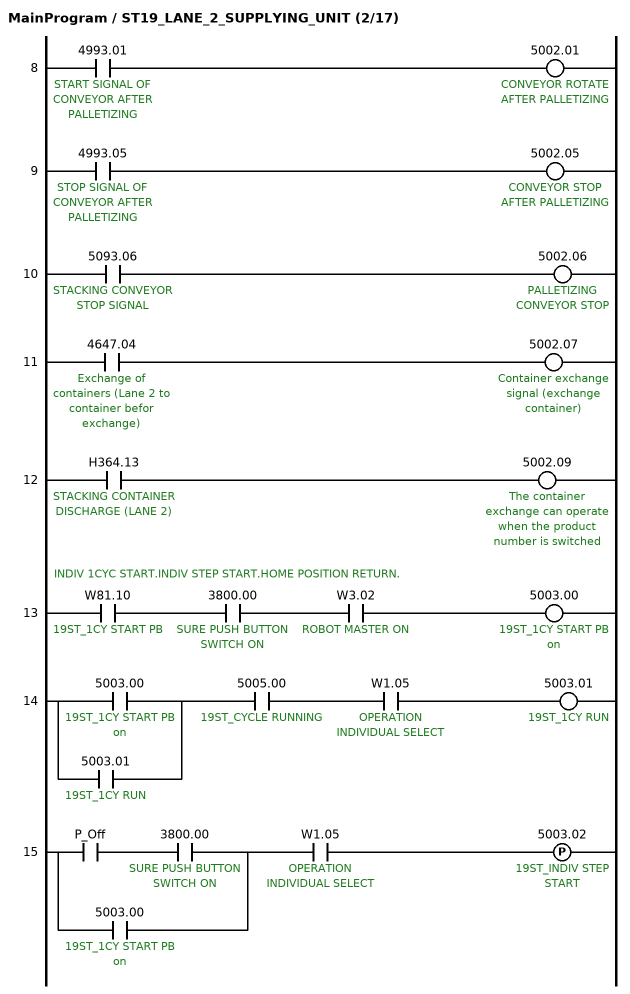
; rung 8
LD 4993.01  ; START SIGNAL OF CONVEYOR AFTER PALLETIZING
OUT 5002.01  ; CONVEYOR ROTATE AFTER PALLETIZING
; rung 9
LD 4993.05  ; STOP SIGNAL OF CONVEYOR AFTER PALLETIZING
OUT 5002.05  ; CONVEYOR STOP AFTER PALLETIZING
; rung 10
LD 5093.06  ; STACKING CONVEYOR STOP SIGNAL
OUT 5002.06  ; PALLETIZING CONVEYOR STOP
; rung 11
LD 4647.04  ; Exchange of containers (Lane 2 to container befor exchange)
OUT 5002.07  ; Container exchange signal (exchange container)
; rung 12
LD H364.13  ; STACKING CONTAINER DISCHARGE (LANE 2)
OUT 5002.09  ; The container exchange can operate when the product number is switched
; rung 13: INDIV 1CYC START.INDIV STEP START.HOME POSITION RETURN.
LD W81.10  ; 19ST_1CY START PB
AND 3800.00  ; SURE PUSH BUTTON SWITCH ON
AND W3.02  ; ROBOT MASTER ON
OUT 5003.00  ; 19ST_1CY START PB on
; rung 14
LD 5003.00  ; 19ST_1CY START PB on
OR 5003.01  ; 19ST_1CY RUN
AND 5005.00  ; 19ST_CYCLE RUNNING
AND W1.05  ; OPERATION INDIVIDUAL SELECT
OUT 5003.01  ; 19ST_1CY RUN
; rung 15
LD P_Off
AND 3800.00  ; SURE PUSH BUTTON SWITCH ON
OR 5003.00  ; 19ST_1CY START PB on
AND W1.05  ; OPERATION INDIVIDUAL SELECT
DIFU(013) 5003.02  ; 19ST_INDIV STEP START

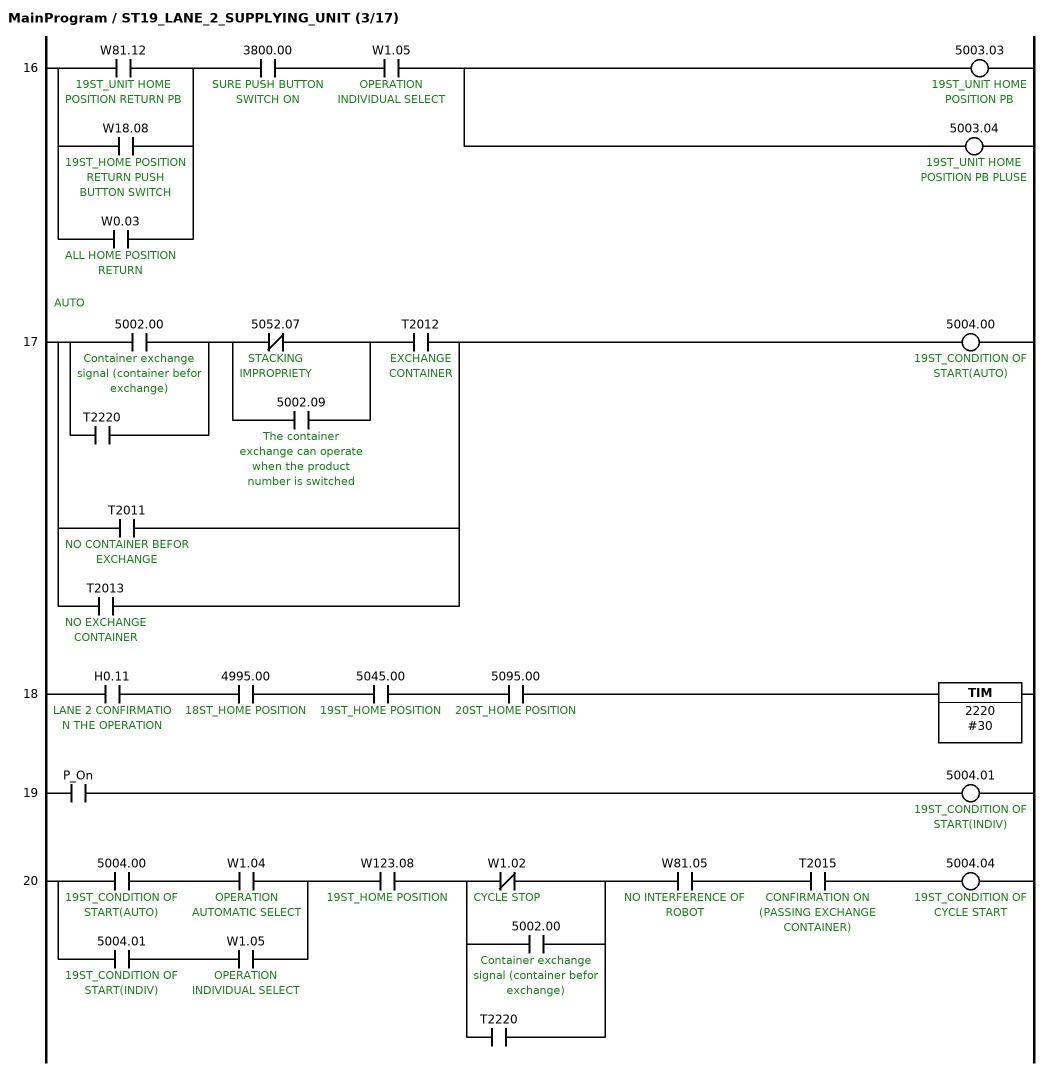
; rung 16
LD W81.12  ; 19ST_UNIT HOME POSITION RETURN PB
OR W18.08  ; 19ST_HOME POSITION RETURN PUSH BUTTON SWITCH
OR W0.03  ; ALL HOME POSITION RETURN
AND 3800.00  ; SURE PUSH BUTTON SWITCH ON
AND W1.05  ; OPERATION INDIVIDUAL SELECT
OUT 5003.03  ; 19ST_UNIT HOME POSITION PB
OUT 5003.04  ; 19ST_UNIT HOME POSITION PB PLUSE
; rung 17: AUTO
LD 5002.00  ; Container exchange signal (container befor exchange)
OR T2220
LDNOT 5052.07  ; STACKING IMPROPRIETY
OR 5002.09  ; The container exchange can operate when the product number is switched
ANDLD
AND T2012  ; EXCHANGE CONTAINER
OR T2011  ; NO CONTAINER BEFOR EXCHANGE
OR T2013  ; NO EXCHANGE CONTAINER
OUT 5004.00  ; 19ST_CONDITION OF START(AUTO)
; rung 18
LD H0.11  ; LANE 2 CONFIRMATION THE OPERATION
AND 4995.00  ; 18ST_HOME POSITION
AND 5045.00  ; 19ST_HOME POSITION
AND 5095.00  ; 20ST_HOME POSITION
TIM 2220 #30
; rung 19
LD P_On
OUT 5004.01  ; 19ST_CONDITION OF START(INDIV)
; rung 20
LD 5004.00  ; 19ST_CONDITION OF START(AUTO)
AND W1.04  ; OPERATION AUTOMATIC SELECT
LD 5004.01  ; 19ST_CONDITION OF START(INDIV)
AND W1.05  ; OPERATION INDIVIDUAL SELECT
ORLD
AND W123.08  ; 19ST_HOME POSITION
LDNOT W1.02  ; CYCLE STOP
OR 5002.00  ; Container exchange signal (container befor exchange)
OR T2220
ANDLD
AND W81.05  ; NO INTERFERENCE OF ROBOT
AND T2015  ; CONFIRMATION ON (PASSING EXCHANGE CONTAINER)
OUT 5004.04  ; 19ST_CONDITION OF CYCLE START

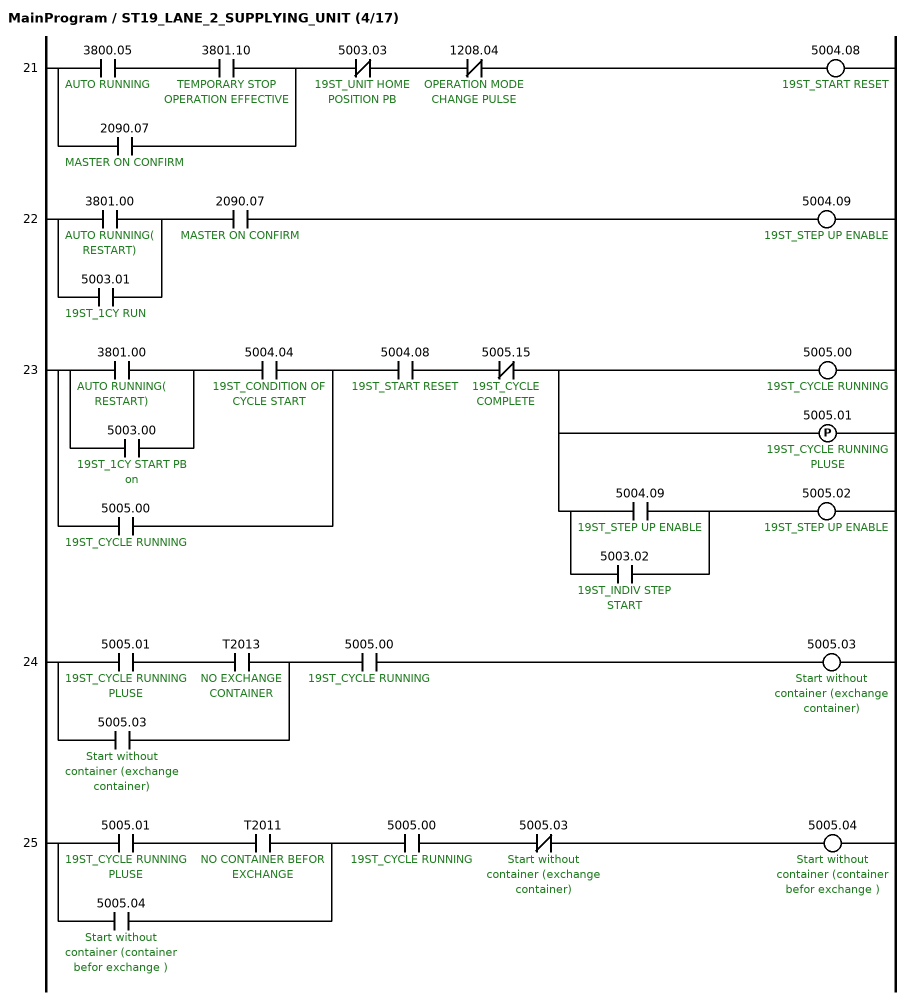
; rung 21
LD 3800.05  ; AUTO RUNNING
AND 3801.10  ; TEMPORARY STOP OPERATION EFFECTIVE
OR 2090.07  ; MASTER ON CONFIRM
ANDNOT 5003.03  ; 19ST_UNIT HOME POSITION PB
ANDNOT 1208.04  ; OPERATION MODE CHANGE PULSE
OUT 5004.08  ; 19ST_START RESET
; rung 22
LD 3801.00  ; AUTO RUNNING(RESTART)
OR 5003.01  ; 19ST_1CY RUN
AND 2090.07  ; MASTER ON CONFIRM
OUT 5004.09  ; 19ST_STEP UP ENABLE
; rung 23
LD 3801.00  ; AUTO RUNNING(RESTART)
OR 5003.00  ; 19ST_1CY START PB on
AND 5004.04  ; 19ST_CONDITION OF CYCLE START
OR 5005.00  ; 19ST_CYCLE RUNNING
AND 5004.08  ; 19ST_START RESET
ANDNOT 5005.15  ; 19ST_CYCLE COMPLETE
OUT 5005.00  ; 19ST_CYCLE RUNNING
DIFU(013) 5005.01  ; 19ST_CYCLE RUNNING PLUSE
LD 5004.09  ; 19ST_STEP UP ENABLE
OR 5003.02  ; 19ST_INDIV STEP START
ANDLD
OUT 5005.02  ; 19ST_STEP UP ENABLE
; rung 24
LD 5005.01  ; 19ST_CYCLE RUNNING PLUSE
AND T2013  ; NO EXCHANGE CONTAINER
OR 5005.03  ; Start without container (exchange container)
AND 5005.00  ; 19ST_CYCLE RUNNING
OUT 5005.03  ; Start without container (exchange container)
; rung 25
LD 5005.01  ; 19ST_CYCLE RUNNING PLUSE
AND T2011  ; NO CONTAINER BEFOR EXCHANGE
OR 5005.04  ; Start without container (container befor exchange )
AND 5005.00  ; 19ST_CYCLE RUNNING
ANDNOT 5005.03  ; Start without container (exchange container)
OUT 5005.04  ; Start without container (container befor exchange )

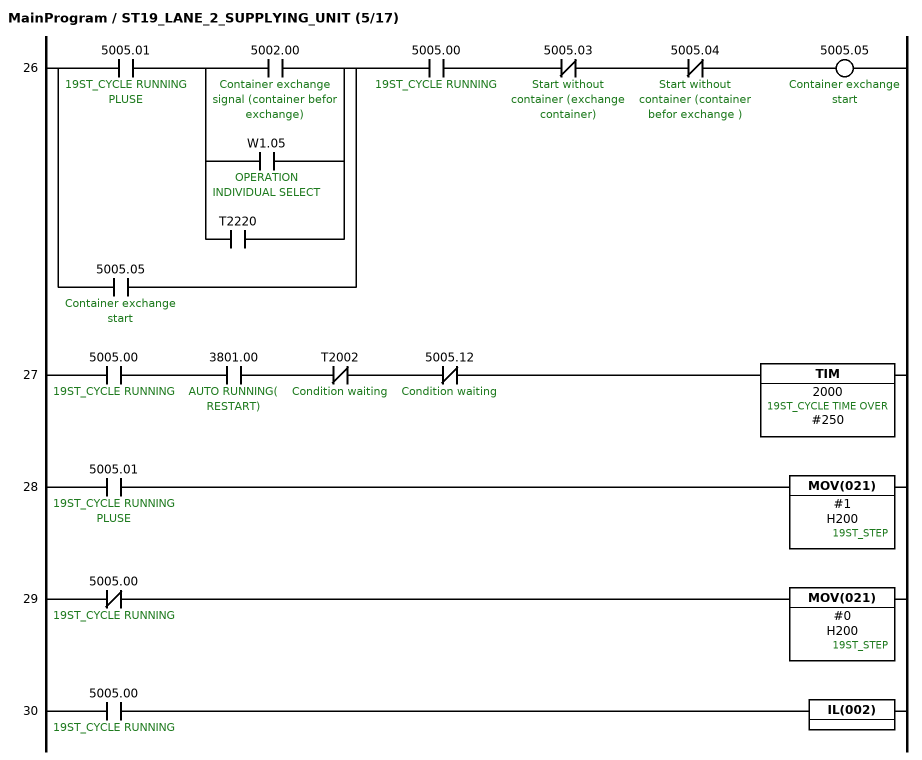
; rung 26
LD 5005.01  ; 19ST_CYCLE RUNNING PLUSE
LD 5002.00  ; Container exchange signal (container befor exchange)
OR W1.05  ; OPERATION INDIVIDUAL SELECT
OR T2220
ANDLD
OR 5005.05  ; Container exchange start
AND 5005.00  ; 19ST_CYCLE RUNNING
ANDNOT 5005.03  ; Start without container (exchange container)
ANDNOT 5005.04  ; Start without container (container befor exchange )
OUT 5005.05  ; Container exchange start
; rung 27
LD 5005.00  ; 19ST_CYCLE RUNNING
AND 3801.00  ; AUTO RUNNING(RESTART)
ANDNOT T2002  ; Condition waiting
ANDNOT 5005.12  ; Condition waiting
TIM 2000 #250  ; 19ST_CYCLE TIME OVER
; rung 28
LD 5005.01  ; 19ST_CYCLE RUNNING PLUSE
MOV(021) #1 H200  ; 19ST_STEP
; rung 29
LDNOT 5005.00  ; 19ST_CYCLE RUNNING
MOV(021) #0 H200  ; 19ST_STEP
; rung 30
LD 5005.00  ; 19ST_CYCLE RUNNING
IL(002)

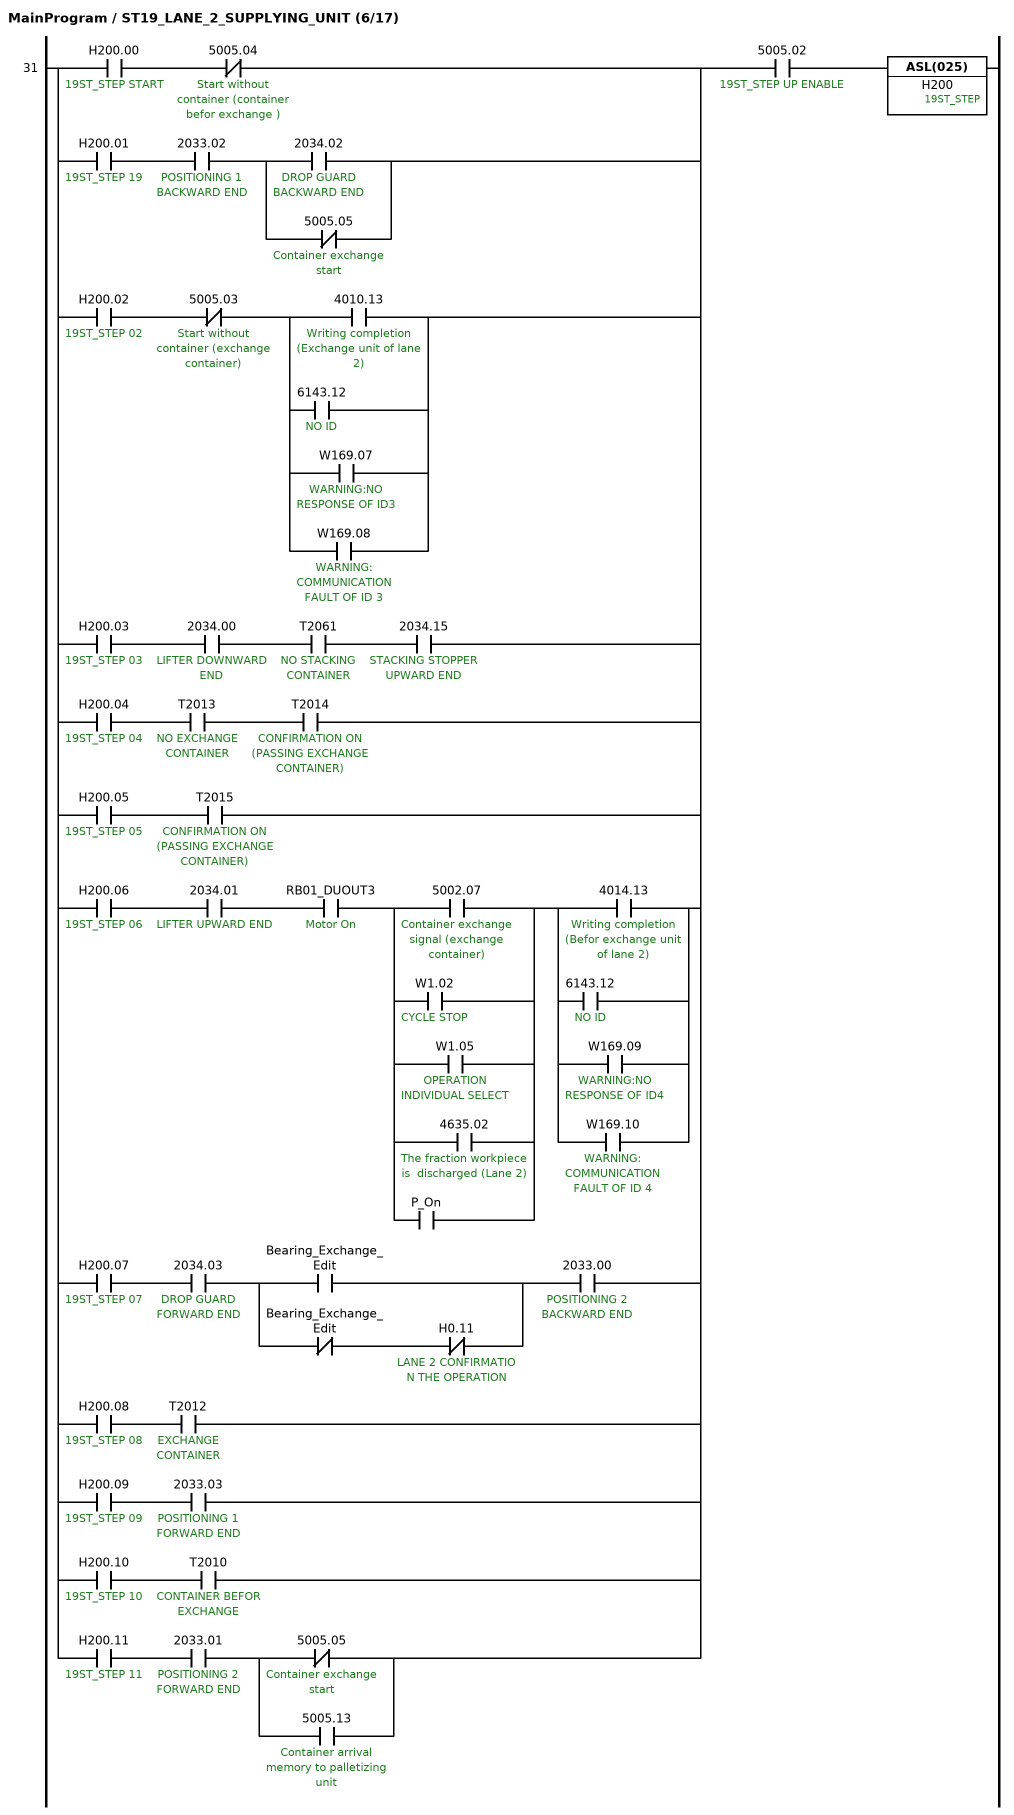
; rung 31
LD H200.00  ; 19ST_STEP START
ANDNOT 5005.04  ; Start without container (container befor exchange )
LD H200.01  ; 19ST_STEP 19
AND 2033.02  ; POSITIONING 1 BACKWARD END
LD 2034.02  ; DROP GUARD BACKWARD END
ORNOT 5005.05  ; Container exchange start
ANDLD
ORLD
LD H200.02  ; 19ST_STEP 02
ANDNOT 5005.03  ; Start without container (exchange container)
LD 4010.13  ; Writing completion (Exchange unit of lane 2)
OR 6143.12  ; NO ID
OR W169.07  ; WARNING:NO RESPONSE OF ID3
OR W169.08  ; WARNING:COMMUNICATION FAULT OF ID 3
ANDLD
ORLD
LD H200.03  ; 19ST_STEP 03
AND 2034.00  ; LIFTER DOWNWARD END
AND T2061  ; NO STACKING CONTAINER
AND 2034.15  ; STACKING STOPPER UPWARD END
ORLD
LD H200.04  ; 19ST_STEP 04
AND T2013  ; NO EXCHANGE CONTAINER
AND T2014  ; CONFIRMATION ON (PASSING EXCHANGE CONTAINER)
ORLD
LD H200.05  ; 19ST_STEP 05
AND T2015  ; CONFIRMATION ON (PASSING EXCHANGE CONTAINER)
ORLD
LD H200.06  ; 19ST_STEP 06
AND 2034.01  ; LIFTER UPWARD END
AND RB01_DUOUT3  ; Motor On
LD 5002.07  ; Container exchange signal (exchange container)
OR W1.02  ; CYCLE STOP
OR W1.05  ; OPERATION INDIVIDUAL SELECT
OR 4635.02  ; The fraction workpiece is  discharged (Lane 2)
OR P_On
ANDLD
LD 4014.13  ; Writing completion (Befor exchange unit of lane 2)
OR 6143.12  ; NO ID
OR W169.09  ; WARNING:NO RESPONSE OF ID4
OR W169.10  ; WARNING:COMMUNICATION FAULT OF ID 4
ANDLD
ORLD
LD H200.07  ; 19ST_STEP 07
AND 2034.03  ; DROP GUARD FORWARD END
LD Bearing_Exchange_Edit
LDNOT Bearing_Exchange_Edit
ANDNOT H0.11  ; LANE 2 CONFIRMATION THE OPERATION
ORLD
ANDLD
AND 2033.00  ; POSITIONING 2 BACKWARD END
ORLD
LD H200.08  ; 19ST_STEP 08
AND T2012  ; EXCHANGE CONTAINER
ORLD
LD H200.09  ; 19ST_STEP 09
AND 2033.03  ; POSITIONING 1 FORWARD END
ORLD
LD H200.10  ; 19ST_STEP 10
AND T2010  ; CONTAINER BEFOR EXCHANGE
ORLD
LD H200.11  ; 19ST_STEP 11
AND 2033.01  ; POSITIONING 2 FORWARD END
LDNOT 5005.05  ; Container exchange start
OR 5005.13  ; Container arrival memory to palletizing unit
ANDLD
ORLD
AND 5005.02  ; 19ST_STEP UP ENABLE
ASL(025) H200  ; 19ST_STEP

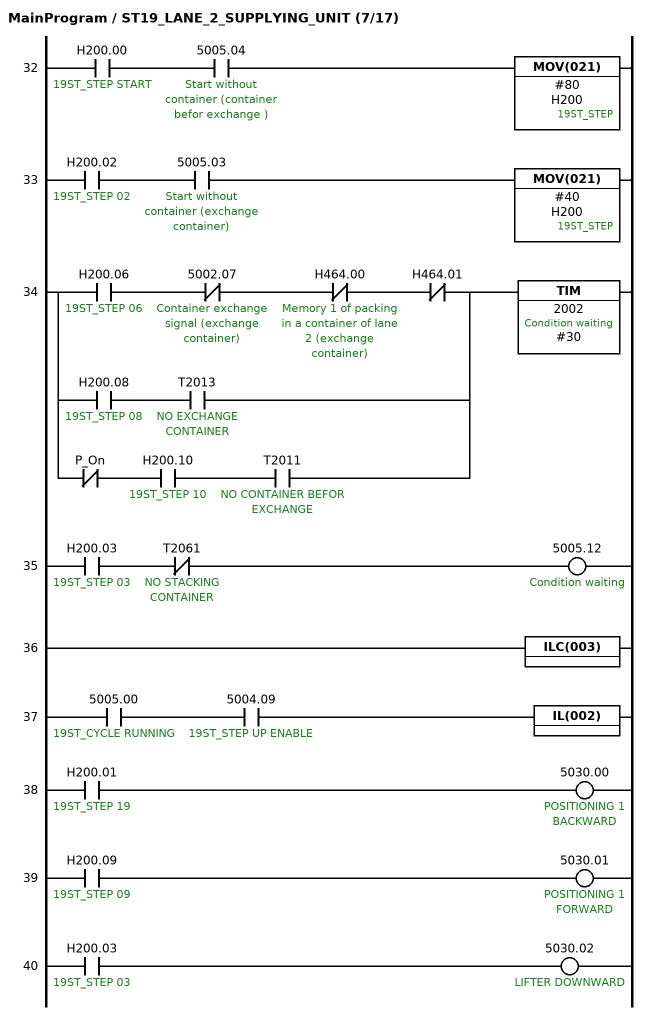
; rung 32
LD H200.00  ; 19ST_STEP START
AND 5005.04  ; Start without container (container befor exchange )
MOV(021) #80 H200  ; 19ST_STEP
; rung 33
LD H200.02  ; 19ST_STEP 02
AND 5005.03  ; Start without container (exchange container)
MOV(021) #40 H200  ; 19ST_STEP
; rung 34
LD H200.06  ; 19ST_STEP 06
ANDNOT 5002.07  ; Container exchange signal (exchange container)
ANDNOT H464.00  ; Memory 1 of packing in a container of lane 2 (exchange container)
ANDNOT H464.01
LD H200.08  ; 19ST_STEP 08
AND T2013  ; NO EXCHANGE CONTAINER
ORLD
LDNOT P_On
AND H200.10  ; 19ST_STEP 10
AND T2011  ; NO CONTAINER BEFOR EXCHANGE
ORLD
TIM 2002 #30  ; Condition waiting
; rung 35
LD H200.03  ; 19ST_STEP 03
ANDNOT T2061  ; NO STACKING CONTAINER
OUT 5005.12  ; Condition waiting
; rung 36
ILC(003)
; rung 37
LD 5005.00  ; 19ST_CYCLE RUNNING
AND 5004.09  ; 19ST_STEP UP ENABLE
IL(002)
; rung 38
LD H200.01  ; 19ST_STEP 19
OUT 5030.00  ; POSITIONING 1 BACKWARD
; rung 39
LD H200.09  ; 19ST_STEP 09
OUT 5030.01  ; POSITIONING 1 FORWARD
; rung 40
LD H200.03  ; 19ST_STEP 03
OUT 5030.02  ; LIFTER DOWNWARD

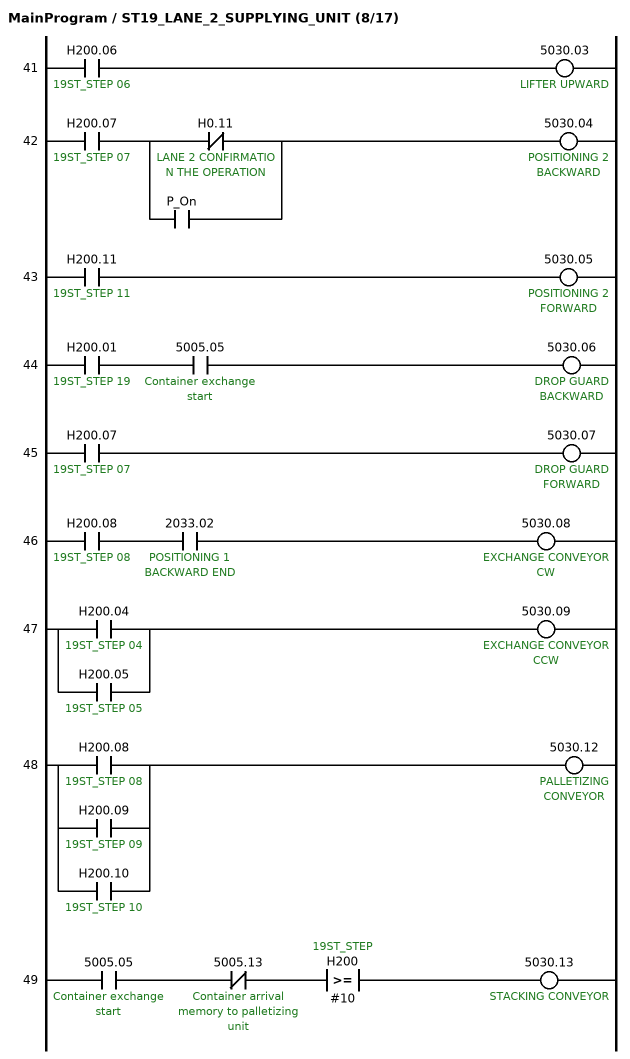
; rung 41
LD H200.06  ; 19ST_STEP 06
OUT 5030.03  ; LIFTER UPWARD
; rung 42
LD H200.07  ; 19ST_STEP 07
LDNOT H0.11  ; LANE 2 CONFIRMATION THE OPERATION
OR P_On
ANDLD
OUT 5030.04  ; POSITIONING 2 BACKWARD
; rung 43
LD H200.11  ; 19ST_STEP 11
OUT 5030.05  ; POSITIONING 2 FORWARD
; rung 44
LD H200.01  ; 19ST_STEP 19
AND 5005.05  ; Container exchange start
OUT 5030.06  ; DROP GUARD BACKWARD
; rung 45
LD H200.07  ; 19ST_STEP 07
OUT 5030.07  ; DROP GUARD FORWARD
; rung 46
LD H200.08  ; 19ST_STEP 08
AND 2033.02  ; POSITIONING 1 BACKWARD END
OUT 5030.08  ; EXCHANGE CONVEYOR CW
; rung 47
LD H200.04  ; 19ST_STEP 04
OR H200.05  ; 19ST_STEP 05
OUT 5030.09  ; EXCHANGE CONVEYOR CCW
; rung 48
LD H200.08  ; 19ST_STEP 08
OR H200.09  ; 19ST_STEP 09
OR H200.10  ; 19ST_STEP 10
OUT 5030.12  ; PALLETIZING CONVEYOR
; rung 49
LD 5005.05  ; Container exchange start
ANDNOT 5005.13  ; Container arrival memory to palletizing unit
AND>=(325) H200 #10  ; 19ST_STEP
OUT 5030.13  ; STACKING CONVEYOR

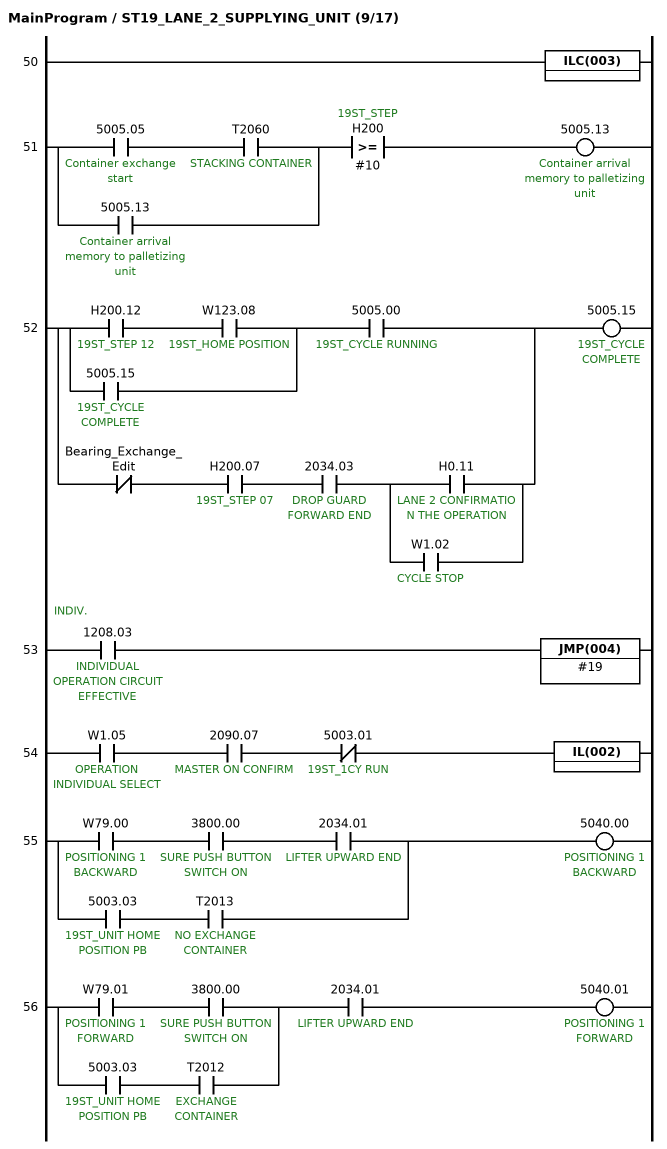
; rung 50
ILC(003)
; rung 51
LD 5005.05  ; Container exchange start
AND T2060  ; STACKING CONTAINER
OR 5005.13  ; Container arrival memory to palletizing unit
AND>=(325) H200 #10  ; 19ST_STEP
OUT 5005.13  ; Container arrival memory to palletizing unit
; rung 52
LD H200.12  ; 19ST_STEP 12
AND W123.08  ; 19ST_HOME POSITION
OR 5005.15  ; 19ST_CYCLE COMPLETE
AND 5005.00  ; 19ST_CYCLE RUNNING
LDNOT Bearing_Exchange_Edit
AND H200.07  ; 19ST_STEP 07
AND 2034.03  ; DROP GUARD FORWARD END
LD H0.11  ; LANE 2 CONFIRMATION THE OPERATION
OR W1.02  ; CYCLE STOP
ANDLD
ORLD
OUT 5005.15  ; 19ST_CYCLE COMPLETE
; rung 53: INDIV.
LD 1208.03  ; INDIVIDUAL OPERATION CIRCUIT EFFECTIVE
JMP(004) #19
; rung 54
LD W1.05  ; OPERATION INDIVIDUAL SELECT
AND 2090.07  ; MASTER ON CONFIRM
ANDNOT 5003.01  ; 19ST_1CY RUN
IL(002)
; rung 55
LD W79.00  ; POSITIONING 1 BACKWARD
AND 3800.00  ; SURE PUSH BUTTON SWITCH ON
AND 2034.01  ; LIFTER UPWARD END
LD 5003.03  ; 19ST_UNIT HOME POSITION PB
AND T2013  ; NO EXCHANGE CONTAINER
ORLD
OUT 5040.00  ; POSITIONING 1 BACKWARD
; rung 56
LD W79.01  ; POSITIONING 1 FORWARD
AND 3800.00  ; SURE PUSH BUTTON SWITCH ON
LD 5003.03  ; 19ST_UNIT HOME POSITION PB
AND T2012  ; EXCHANGE CONTAINER
ORLD
AND 2034.01  ; LIFTER UPWARD END
OUT 5040.01  ; POSITIONING 1 FORWARD

